KUKA KRL program: EPS_2_251825_SA27_A_20260116064105.src

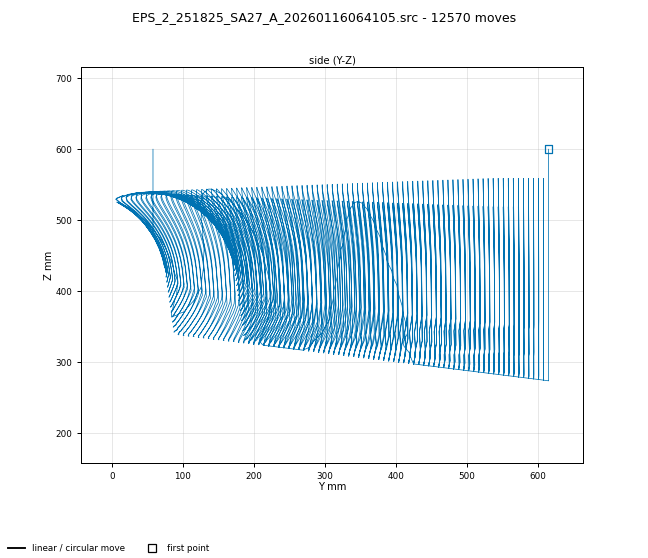
[picture p0: tool path of EPS_2_251825_SA27_A_20260116064105.src, 12570 of 12572 moves have a stored position in this frame; points joined in program order, loops and branches not executed]
&ACCESS RVP
&REL 4
&COMMENT QRS 19112012
&PARAM EDITMASK = *
DEF PART()
EXT BAS (BAS_COMMAND :IN,REAL :IN )
INT I
BAS (#INITMOV,0 )

;KUKA QRS Post kuka4.cps  Date:22-06-2017 !

File_ID=2986

QRS_PRE_INIT()

;Init var - Until changes are made in qrs_pre_init
Outlet_Square_prg=0
Inlet_1_Square_prg=0
Inlet_2_Square_prg=0
Inlet_3_Square_prg=0
Inlet_4_Square_prg=0
Inlet_5_Square_prg=0

Outlet_1={X 0.000, Y 535.490, Z 458.500, B 0.000, E1 0.000 }
Inlet_1={X 0.000, Y 538.340, Z 418.500, B 0.000, E1 212.000 }
Outlet_1_type=201
Inlet_1_type=201
;QRS#1=Sidecore dimensions
;QRS#2=200-8" PVC SDR 35
;QRS#3=200-8" PVC SDR 35
;QRS#4=
;QRS#5=
;QRS#6=
;QRS#7=
;QRS#8=
;QRS#9=12-08 PSX
;QRS#10=12-08 PSX
;QRS#11=
;QRS#12=
;QRS#13=
;QRS#14=
;QRS#15=
;QRS#16=1220x127x838 2,75'
;QRS#17=EPS Height
;QRS#18=559
;QRS#19=*
;QRS#20= UPDATED VERSION 22-06-2017
;QRS#21=*
Outlet_Square=0100
Inlet_1_Square=0100
Inlet_2_Square=0
Inlet_3_Square=0
Inlet_4_Square=0
Inlet_5_Square=0
Mill_Square=1
Outlet_Square_Prg=204
Inlet_1_Square_prg=204

QRS_INIT()

$ADVANCE=5

; T1
PTP {E1 173.63,E2 173.63}
PTP {X 0,Y 615.439,A -85,B 0,C 180,E1 173.63,E2 173.63,E3 0,E4 0,E5 0,E6 0}
QRS_SPEED_INIT()
LIN {X 0,Y 615.439,Z 600,A -85,B 0,C 180,E1 173.63,E2 173.63,E3 0,E4 0,E5 0,E6 0} C_VEL
LIN {X 0,Y 615.439,Z 283.873,A -85,B 0,C 180,E1 173.63,E2 173.63} C_VEL
LIN {X 0,Y 615.439,Z 275.692,A -85,B 0,C 180,E1 173.63,E2 173.63} C_VEL
LIN {X 0,Y 615.44,Z 273.692,A -85,B 0,C 180,E1 173.444,E2 173.444} C_VEL
LIN {X 0,Y 615.485,Z 273.687,A -85,B 0,C 180,E1 170.801,E2 170.801} C_VEL
LIN {X 0,Y 615.48,Z 273.701,A -85,B 0,C 180,E1 168.139,E2 168.139} C_VEL
LIN {X 0,Y 615.434,Z 273.695,A -85,B 0,C 180,E1 165.45,E2 165.45} C_VEL
LIN {X 0,Y 615.431,Z 273.695,A -85,B 0,C 180,E1 163.412,E2 163.412} C_VEL
LIN {X 0,Y 615.431,Z 273.695,A -85,B 0,C 180,E1 161.352,E2 161.352} C_VEL
LIN {X 0,Y 615.429,Z 273.695,A -85,B 0,C 180,E1 159.267,E2 159.267} C_VEL
LIN {X 0,Y 615.427,Z 273.695,A -85,B 0,C 180,E1 157.153,E2 157.153} C_VEL
LIN {X 0,Y 615.424,Z 273.695,A -85,B 0,C 180,E1 155.005,E2 155.005} C_VEL
LIN {X 0,Y 615.425,Z 273.695,A -85,B 0,C 180,E1 152.82,E2 152.82} C_VEL
LIN {X 0,Y 615.469,Z 273.693,A -85,B 0,C 180,E1 150.206,E2 150.206} C_VEL
LIN {X 0,Y 615.469,Z 273.699,A -85,B 0,C 180,E1 147.541,E2 147.541} C_VEL
LIN {X 0,Y 615.434,Z 273.698,A -85,B 0,C 180,E1 145.181,E2 145.181} C_VEL
LIN {X 0,Y 615.415,Z 273.698,A -85,B 0,C 180,E1 142.752,E2 142.752} C_VEL
LIN {X 0,Y 615.46,Z 273.696,A -85,B 0,C 180,E1 139.913,E2 139.913} C_VEL
LIN {X 0,Y 615.489,Z 273.697,A -85,B 0,C 180,E1 137.647,E2 137.647} C_VEL
LIN {X 0,Y 615.426,Z 273.7,A -85,B 0,C 180,E1 134.925,E2 134.925} C_VEL
LIN {X 0,Y 615.445,Z 273.7,A -85,B 0,C 180,E1 133.043,E2 133.043} C_VEL
LIN {X 0,Y 615.41,Z 273.7,A -85,B 0,C 180,E1 130.612,E2 130.612} C_VEL
LIN {X 0,Y 615.407,Z 273.7,A -85,B 0,C 180,E1 128.074,E2 128.074} C_VEL
LIN {X 0,Y 615.435,Z 273.701,A -85,B 0,C 180,E1 125.619,E2 125.619} C_VEL
LIN {X 0,Y 615.47,Z 273.704,A -85,B 0,C 180,E1 123.237,E2 123.237} C_VEL
LIN {X 0,Y 615.472,Z 273.699,A -85,B 0,C 180,E1 120.921,E2 120.921} C_VEL
LIN {X 0,Y 615.431,Z 273.697,A -85,B 0,C 180,E1 118.44,E2 118.44} C_VEL
LIN {X 0,Y 615.434,Z 273.697,A -85,B 0,C 180,E1 116.447,E2 116.447} C_VEL
LIN {X 0,Y 615.427,Z 273.697,A -85,B 0,C 180,E1 114.275,E2 114.275} C_VEL
LIN {X 0,Y 615.427,Z 273.696,A -85,B 0,C 180,E1 112.139,E2 112.139} C_VEL
LIN {X 0,Y 615.426,Z 273.695,A -85,B 0,C 180,E1 110.036,E2 110.036} C_VEL
LIN {X 0,Y 615.427,Z 273.695,A -85,B 0,C 180,E1 107.96,E2 107.96} C_VEL
LIN {X 0,Y 615.429,Z 273.695,A -85,B 0,C 180,E1 105.908,E2 105.908} C_VEL
LIN {X 0,Y 615.432,Z 273.694,A -85,B 0,C 180,E1 103.877,E2 103.877} C_VEL
LIN {X 0,Y 615.437,Z 273.693,A -85,B 0,C 180,E1 101.863,E2 101.863} C_VEL
LIN {X 0,Y 615.443,Z 273.692,A -85,B 0,C 180,E1 99.864,E2 99.864} C_VEL
LIN {X 0,Y 615.448,Z 273.692,A -85,B 0,C 180,E1 97.878,E2 97.878} C_VEL
LIN {X 0,Y 615.46,Z 273.69,A -85,B 0,C 180,E1 95.901,E2 95.901} C_VEL
LIN {X 0,Y 615.432,Z 273.694,A -85,B 0,C 180,E1 93.275,E2 93.275} C_VEL
LIN {X 0,Y 615.464,Z 273.698,A -85,B 0,C 180,E1 90.656,E2 90.656} C_VEL
LIN {X 0,Y 615.497,Z 273.69,A -85,B 0,C 180,E1 88.039,E2 88.039} C_VEL
LIN {X 0,Y 615.451,Z 273.69,A -85,B 0,C 180,E1 85.418,E2 85.418} C_VEL
LIN {X 0,Y 615.456,Z 273.689,A -85,B 0,C 180,E1 83.446,E2 83.446} C_VEL
LIN {X 0,Y 615.468,Z 273.687,A -85,B 0,C 180,E1 81.466,E2 81.466} C_VEL
LIN {X 0,Y 615.449,Z 273.689,A -85,B 0,C 180,E1 79.132,E2 79.132} C_VEL
LIN {X 0,Y 615.448,Z 273.76,A -85,B 0,C 180,E1 76.612,E2 76.612} C_VEL
LIN {X 0,Y 615.487,Z 288.561,A -85,B 0,C 180,E1 74.098,E2 74.098} C_VEL
LIN {X 0,Y 615.49,Z 304.913,A -85,B 0,C 180,E1 71.358,E2 71.358} C_VEL
LIN {X 0,Y 615.481,Z 308.156,A -85,B 0,C 180,E1 70.817,E2 70.817} C_VEL
LIN {X 0,Y 615.479,Z 414.874,A -85,B 0,C 180,E1 69.544,E2 69.544} C_VEL
LIN {X 0,Y 615.49,Z 427.341,A -85,B 0,C 180,E1 69.273,E2 69.273} C_VEL
LIN {X 0,Y 615.492,Z 439.612,A -85,B 0,C 180,E1 68.879,E2 68.879} C_VEL
LIN {X 0,Y 615.472,Z 450.84,A -85,B 0,C 180,E1 68.396,E2 68.396} C_VEL
LIN {X 0,Y 615.466,Z 462.297,A -85,B 0,C 180,E1 67.762,E2 67.762} C_VEL
LIN {X 0,Y 615.498,Z 473.358,A -85,B 0,C 180,E1 66.982,E2 66.982} C_VEL
LIN {X 0,Y 615.498,Z 482.093,A -85,B 0,C 180,E1 66.219,E2 66.219} C_VEL
LIN {X 0,Y 615.497,Z 490.274,A -85,B 0,C 180,E1 65.373,E2 65.373} C_VEL
LIN {X 0,Y 615.493,Z 497.637,A -85,B 0,C 180,E1 64.431,E2 64.431} C_VEL
LIN {X 0,Y 615.497,Z 503.202,A -85,B 0,C 180,E1 63.561,E2 63.561} C_VEL
LIN {X 0,Y 615.496,Z 508.785,A -85,B 0,C 180,E1 62.459,E2 62.459} C_VEL
LIN {X 0,Y 615.496,Z 513.017,A -85,B 0,C 180,E1 61.347,E2 61.347} C_VEL
LIN {X 0,Y 615.496,Z 516.043,A -85,B 0,C 180,E1 60.205,E2 60.205} C_VEL
LIN {X 0,Y 615.497,Z 517.96,A -85,B 0,C 180,E1 58.913,E2 58.913} C_VEL
LIN {X 0,Y 615.494,Z 518.326,A -85,B 0,C 180,E1 57.669,E2 57.669} C_VEL
LIN {X 0,Y 615.496,Z 517.367,A -85,B 0,C 180,E1 56.465,E2 56.465} C_VEL
LIN {X 0,Y 615.492,Z 514.843,A -85,B 0,C 180,E1 55.191,E2 55.191} C_VEL
LIN {X 0,Y 615.495,Z 511.661,A -85,B 0,C 180,E1 54.166,E2 54.166} C_VEL
LIN {X 0,Y 615.492,Z 506.976,A -85,B 0,C 180,E1 53.063,E2 53.063} C_VEL
LIN {X 0,Y 615.495,Z 500.7,A -85,B 0,C 180,E1 51.938,E2 51.938} C_VEL
LIN {X 0,Y 615.496,Z 493.587,A -85,B 0,C 180,E1 50.937,E2 50.937} C_VEL
LIN {X 0,Y 615.497,Z 486.114,A -85,B 0,C 180,E1 50.084,E2 50.084} C_VEL
LIN {X 0,Y 615.495,Z 476.164,A -85,B 0,C 180,E1 49.153,E2 49.153} C_VEL
LIN {X 0,Y 615.481,Z 465.87,A -85,B 0,C 180,E1 48.381,E2 48.381} C_VEL
LIN {X 0,Y 615.459,Z 454.84,A -85,B 0,C 180,E1 47.719,E2 47.719} C_VEL
LIN {X 0,Y 615.495,Z 442.203,A -85,B 0,C 180,E1 47.129,E2 47.129} C_VEL
LIN {X 0,Y 615.492,Z 430.199,A -85,B 0,C 180,E1 46.715,E2 46.715} C_VEL
LIN {X 0,Y 615.482,Z 417.178,A -85,B 0,C 180,E1 46.409,E2 46.409} C_VEL
LIN {X 0,Y 615.471,Z 395.409,A -85,B 0,C 180,E1 46.124,E2 46.124} C_VEL
LIN {X 0,Y 615.482,Z 308.164,A -85,B 0,C 180,E1 45.094,E2 45.094} C_VEL
LIN {X 0,Y 615.496,Z 291.775,A -85,B 0,C 180,E1 42.353,E2 42.353} C_VEL
LIN {X 0,Y 615.465,Z 275.402,A -85,B 0,C 180,E1 39.579,E2 39.579} C_VEL
LIN {X 0,Y 615.445,Z 273.695,A -85,B 0,C 180,E1 39.279,E2 39.279} C_VEL
LIN {X 0,Y 615.439,Z 273.692,A -85,B 0,C 180,E1 36.939,E2 36.939} C_VEL
LIN {X 0,Y 615.443,Z 273.691,A -85,B 0,C 180,E1 34.704,E2 34.704} C_VEL
LIN {X 0,Y 615.465,Z 273.69,A -85,B 0,C 180,E1 32.338,E2 32.338} C_VEL
LIN {X 0,Y 615.463,Z 273.698,A -85,B 0,C 180,E1 29.408,E2 29.408} C_VEL
LIN {X 0,Y 615.434,Z 273.697,A -85,B 0,C 180,E1 27.048,E2 27.048} C_VEL
LIN {X 0,Y 615.432,Z 273.697,A -85,B 0,C 180,E1 24.994,E2 24.994} C_VEL
LIN {X 0,Y 615.425,Z 273.697,A -85,B 0,C 180,E1 22.847,E2 22.847} C_VEL
LIN {X 0,Y 615.418,Z 273.697,A -85,B 0,C 180,E1 20.556,E2 20.556} C_VEL
LIN {X 0,Y 615.446,Z 273.696,A -85,B 0,C 180,E1 17.958,E2 17.958} C_VEL
LIN {X 0,Y 615.469,Z 273.7,A -85,B 0,C 180,E1 15.227,E2 15.227} C_VEL
LIN {X 0,Y 615.409,Z 273.699,A -85,B 0,C 180,E1 12.532,E2 12.532} C_VEL
LIN {X 0,Y 615.408,Z 273.7,A -85,B 0,C 180,E1 10.528,E2 10.528} C_VEL
LIN {X 0,Y 615.41,Z 273.7,A -85,B 0,C 180,E1 8.538,E2 8.538} C_VEL
LIN {X 0,Y 615.416,Z 273.699,A -85,B 0,C 180,E1 6.557,E2 6.557} C_VEL
LIN {X 0,Y 615.423,Z 273.699,A -85,B 0,C 180,E1 4.585,E2 4.585} C_VEL
LIN {X 0,Y 615.434,Z 273.697,A -85,B 0,C 180,E1 2.618,E2 2.618} C_VEL
LIN {X 0,Y 615.442,Z 273.697,A -85,B 0,C 180,E1 0.654,E2 0.654} C_VEL
LIN {X 0,Y 615.417,Z 273.697,A -85,B 0,C 180,E1 -1.963,E2 -1.963} C_VEL
LIN {X 0,Y 615.419,Z 273.697,A -85,B 0,C 180,E1 -3.929,E2 -3.929} C_VEL
LIN {X 0,Y 615.426,Z 273.695,A -85,B 0,C 180,E1 -5.899,E2 -5.899} C_VEL
LIN {X 0,Y 615.432,Z 273.694,A -85,B 0,C 180,E1 -7.876,E2 -7.876} C_VEL
LIN {X 0,Y 615.438,Z 273.693,A -85,B 0,C 180,E1 -9.863,E2 -9.863} C_VEL
LIN {X 0,Y 615.443,Z 273.692,A -85,B 0,C 180,E1 -11.862,E2 -11.862} C_VEL
LIN {X 0,Y 615.444,Z 273.692,A -85,B 0,C 180,E1 -13.941,E2 -13.941} C_VEL
LIN {X 0,Y 615.454,Z 273.69,A -85,B 0,C 180,E1 -15.906,E2 -15.906} C_VEL
LIN {X 0,Y 615.456,Z 273.689,A -85,B 0,C 180,E1 -17.958,E2 -17.958} C_VEL
LIN {X 0,Y 615.457,Z 273.689,A -85,B 0,C 180,E1 -20.034,E2 -20.034} C_VEL
LIN {X 0,Y 615.445,Z 273.691,A -85,B 0,C 180,E1 -22.351,E2 -22.351} C_VEL
LIN {X 0,Y 615.452,Z 273.689,A -85,B 0,C 180,E1 -24.274,E2 -24.274} C_VEL
LIN {X 0,Y 615.448,Z 273.69,A -85,B 0,C 180,E1 -26.446,E2 -26.446} C_VEL
LIN {X 0,Y 615.449,Z 273.691,A -85,B 0,C 180,E1 -28.66,E2 -28.66} C_VEL
LIN {X 0,Y 615.464,Z 273.696,A -85,B 0,C 180,E1 -31.093,E2 -31.093} C_VEL
LIN {X 0,Y 615.494,Z 273.684,A -85,B 0,C 180,E1 -34.022,E2 -34.022} C_VEL
LIN {X 0,Y 615.477,Z 273.684,A -85,B 0,C 180,E1 -36.426,E2 -36.426} C_VEL
LIN {X 0,Y 615.461,Z 273.692,A -85,B 0,C 180,E1 -39.067,E2 -39.067} C_VEL
LIN {X 0,Y 615.477,Z 273.699,A -85,B 0,C 180,E1 -41.475,E2 -41.475} C_VEL
LIN {X 0,Y 615.484,Z 273.688,A -85,B 0,C 180,E1 -44.15,E2 -44.15} C_VEL
LIN {X 0,Y 615.47,Z 273.686,A -85,B 0,C 180,E1 -46.955,E2 -46.955} C_VEL
LIN {X 0,Y 615.471,Z 273.693,A -85,B 0,C 180,E1 -49.399,E2 -49.399} C_VEL
LIN {X 0,Y 615.489,Z 273.697,A -85,B 0,C 180,E1 -51.988,E2 -51.988} C_VEL
LIN {X 0,Y 615.476,Z 273.689,A -85,B 0,C 180,E1 -54.389,E2 -54.389} C_VEL
LIN {X 0,Y 615.483,Z 273.683,A -85,B 0,C 180,E1 -56.769,E2 -56.769} C_VEL
LIN {X 0,Y 615.483,Z 273.682,A -85,B 0,C 180,E1 -59.085,E2 -59.085} C_VEL
LIN {X 0,Y 615.477,Z 273.69,A -85,B 0,C 180,E1 -61.552,E2 -61.552} C_VEL
LIN {X 0,Y 615.481,Z 273.696,A -85,B 0,C 180,E1 -64.288,E2 -64.288} C_VEL
LIN {X 0,Y 615.489,Z 273.681,A -85,B 0,C 180,E1 -67.16,E2 -67.16} C_VEL
LIN {X 0,Y 615.487,Z 273.766,A -85,B 0,C 180,E1 -67.439,E2 -67.439} C_VEL
LIN {X 0,Y 615.456,Z 293.719,A -85,B 0,C 180,E1 -70.144,E2 -70.144} C_VEL
LIN {X 0,Y 615.472,Z 313.103,A -85,B 0,C 180,E1 -72.733,E2 -72.733} C_VEL
LIN {X 0,Y 615.493,Z 334.935,A -85,B 0,C 180,E1 -75.609,E2 -75.609} C_VEL
LIN {X 0,Y 615.471,Z 346.492,A -85,B 0,C 180,E1 -77.116,E2 -77.116} C_VEL
LIN {X 0,Y 615.457,Z 455.001,A -85,B 0,C 180,E1 -78.413,E2 -78.413} C_VEL
LIN {X 0,Y 615.456,Z 467.457,A -85,B 0,C 180,E1 -78.684,E2 -78.684} C_VEL
LIN {X 0,Y 615.483,Z 480.688,A -85,B 0,C 180,E1 -79.116,E2 -79.116} C_VEL
LIN {X 0,Y 615.492,Z 492.532,A -85,B 0,C 180,E1 -79.642,E2 -79.642} C_VEL
LIN {X 0,Y 615.483,Z 504.039,A -85,B 0,C 180,E1 -80.307,E2 -80.307} C_VEL
LIN {X 0,Y 615.499,Z 514.376,A -85,B 0,C 180,E1 -81.053,E2 -81.053} C_VEL
LIN {X 0,Y 615.497,Z 522.719,A -85,B 0,C 180,E1 -81.797,E2 -81.797} C_VEL
LIN {X 0,Y 615.498,Z 530.629,A -85,B 0,C 180,E1 -82.622,E2 -82.622} C_VEL
LIN {X 0,Y 615.491,Z 538.221,A -85,B 0,C 180,E1 -83.611,E2 -83.611} C_VEL
LIN {X 0,Y 615.498,Z 545.218,A -85,B 0,C 180,E1 -84.761,E2 -84.761} C_VEL
LIN {X 0,Y 615.493,Z 549.862,A -85,B 0,C 180,E1 -85.746,E2 -85.746} C_VEL
LIN {X 0,Y 615.494,Z 553.406,A -85,B 0,C 180,E1 -86.729,E2 -86.729} C_VEL
LIN {X 0,Y 615.497,Z 555.239,A -85,B 0,C 180,E1 -87.384,E2 -87.384} C_VEL
LIN {X 0,Y 615.497,Z 556.612,A -85,B 0,C 180,E1 -88.039,E2 -88.039} C_VEL
LIN {X 0,Y 615.496,Z 558.175,A -85,B 0,C 180,E1 -89.348,E2 -89.348} C_VEL
LIN {X 0,Y 615.494,Z 558.389,A -85,B 0,C 180,E1 -90.002,E2 -90.002} C_VEL
LIN {X 0,Y 615.495,Z 557.578,A -85,B 0,C 180,E1 -91.311,E2 -91.311} C_VEL
LIN {X 0,Y 615.497,Z 556.605,A -85,B 0,C 180,E1 -91.965,E2 -91.965} C_VEL
LIN {X 0,Y 615.497,Z 555.228,A -85,B 0,C 180,E1 -92.62,E2 -92.62} C_VEL
LIN {X 0,Y 615.496,Z 552.343,A -85,B 0,C 180,E1 -93.603,E2 -93.603} C_VEL
LIN {X 0,Y 615.498,Z 548.434,A -85,B 0,C 180,E1 -94.586,E2 -94.586} C_VEL
LIN {X 0,Y 615.499,Z 543.395,A -85,B 0,C 180,E1 -95.571,E2 -95.571} C_VEL
LIN {X 0,Y 615.49,Z 536.913,A -85,B 0,C 180,E1 -96.578,E2 -96.578} C_VEL
LIN {X 0,Y 615.497,Z 529.118,A -85,B 0,C 180,E1 -97.547,E2 -97.547} C_VEL
LIN {X 0,Y 615.498,Z 519.239,A -85,B 0,C 180,E1 -98.538,E2 -98.538} C_VEL
LIN {X 0,Y 615.495,Z 508.845,A -85,B 0,C 180,E1 -99.366,E2 -99.366} C_VEL
LIN {X 0,Y 615.482,Z 498.551,A -85,B 0,C 180,E1 -100.03,E2 -100.03} C_VEL
LIN {X 0,Y 615.495,Z 487.113,A -85,B 0,C 180,E1 -100.617,E2 -100.617} C_VEL
LIN {X 0,Y 615.466,Z 475.331,A -85,B 0,C 180,E1 -101.079,E2 -101.079} C_VEL
LIN {X 0,Y 615.455,Z 462.187,A -85,B 0,C 180,E1 -101.445,E2 -101.445} C_VEL
LIN {X 0,Y 615.461,Z 448.837,A -85,B 0,C 180,E1 -101.675,E2 -101.675} C_VEL
LIN {X 0,Y 615.471,Z 346.459,A -85,B 0,C 180,E1 -102.888,E2 -102.888} C_VEL
LIN {X 0,Y 615.455,Z 325.982,A -85,B 0,C 180,E1 -105.567,E2 -105.567} C_VEL
LIN {X 0,Y 615.481,Z 305.471,A -85,B 0,C 180,E1 -108.282,E2 -108.282} C_VEL
LIN {X 0,Y 615.468,Z 283.338,A -85,B 0,C 180,E1 -111.258,E2 -111.258} C_VEL
LIN {X 0,Y 615.489,Z 273.682,A -85,B 0,C 180,E1 -112.594,E2 -112.594} C_VEL
LIN {X 0,Y 615.485,Z 273.681,A -85,B 0,C 180,E1 -114.992,E2 -114.992} C_VEL
LIN {X 0,Y 615.481,Z 273.7,A -85,B 0,C 180,E1 -117.916,E2 -117.916} C_VEL
LIN {X 0,Y 615.492,Z 273.698,A -85,B 0,C 180,E1 -120.16,E2 -120.16} C_VEL
LIN {X 0,Y 615.479,Z 273.692,A -85,B 0,C 180,E1 -122.458,E2 -122.458} C_VEL
LIN {X 0,Y 615.478,Z 273.686,A -85,B 0,C 180,E1 -124.815,E2 -124.815} C_VEL
LIN {X 0,Y 615.49,Z 273.68,A -85,B 0,C 180,E1 -127.242,E2 -127.242} C_VEL
LIN {X 0,Y 615.484,Z 273.695,A -85,B 0,C 180,E1 -130.088,E2 -130.088} C_VEL
LIN {X 0,Y 615.499,Z 273.7,A -85,B 0,C 180,E1 -132.351,E2 -132.351} C_VEL
LIN {X 0,Y 615.472,Z 273.687,A -85,B 0,C 180,E1 -135.069,E2 -135.069} C_VEL
LIN {X 0,Y 615.482,Z 273.686,A -85,B 0,C 180,E1 -137.919,E2 -137.919} C_VEL
LIN {X 0,Y 615.483,Z 273.693,A -85,B 0,C 180,E1 -140.249,E2 -140.249} C_VEL
LIN {X 0,Y 615.467,Z 273.692,A -85,B 0,C 180,E1 -143.064,E2 -143.064} C_VEL
LIN {X 0,Y 615.466,Z 273.689,A -85,B 0,C 180,E1 -145.3,E2 -145.3} C_VEL
LIN {X 0,Y 615.476,Z 273.683,A -85,B 0,C 180,E1 -147.669,E2 -147.669} C_VEL
LIN {X 0,Y 615.486,Z 273.696,A -85,B 0,C 180,E1 -150.594,E2 -150.594} C_VEL
LIN {X 0,Y 615.488,Z 273.698,A -85,B 0,C 180,E1 -152.952,E2 -152.952} C_VEL
LIN {X 0,Y 615.463,Z 273.687,A -85,B 0,C 180,E1 -155.727,E2 -155.727} C_VEL
LIN {X 0,Y 615.488,Z 273.688,A -85,B 0,C 180,E1 -158.568,E2 -158.568} C_VEL
LIN {X 0,Y 615.466,Z 273.695,A -85,B 0,C 180,E1 -161.396,E2 -161.396} C_VEL
LIN {X 0,Y 615.464,Z 273.686,A -85,B 0,C 180,E1 -164.094,E2 -164.094} C_VEL
LIN {X 0,Y 615.491,Z 273.689,A -85,B 0,C 180,E1 -166.799,E2 -166.799} C_VEL
LIN {X 0,Y 615.473,Z 273.697,A -85,B 0,C 180,E1 -169.473,E2 -169.473} C_VEL
LIN {X 0,Y 615.45,Z 273.69,A -85,B 0,C 180,E1 -172.124,E2 -172.124} C_VEL
LIN {X 0,Y 615.486,Z 273.685,A -85,B 0,C 180,E1 -174.759,E2 -174.759} C_VEL
LIN {X 0,Y 615.497,Z 273.699,A -85,B 0,C 180,E1 -177.382,E2 -177.382} C_VEL
LIN {X 0,Y 615.448,Z 273.695,A -85,B 0,C 180,E1 -180,E2 -180} C_VEL
LIN {X 0,Y 615.454,Z 273.696,A -85,B 0,C 180,E1 -181.963,E2 -181.963} C_VEL
LIN {X 0,Y 615.459,Z 273.697,A -85,B 0,C 180,E1 -183.929,E2 -183.929} C_VEL
LIN {X 0,Y 615.466,Z 273.698,A -85,B 0,C 180,E1 -185.899,E2 -185.899} C_VEL
LIN {X 0,Y 615.44,Z 273.692,A -85,B 0,C 180,E1 -186.556,E2 -186.556} C_VEL
LIN {X 0,Y 614.8,Z 273.837,A -85,B 0,C 180,E1 -187.102,E2 -187.102} C_VEL
LIN {X 0,Y 611.989,Z 274.252,A -85,B 0,C 180,E1 -187.988,E2 -187.988} C_VEL
LIN {X 0,Y 609.593,Z 274.561,A -85,B 0,C 180,E1 -188.701,E2 -188.701} C_VEL
LIN {X 0,Y 608.548,Z 274.68,A -85,B 0,C 180,E1 -189.25,E2 -189.25} C_VEL
LIN {X 0,Y 608.455,Z 274.69,A -85,B 0,C 180,E1 -189.437,E2 -189.437} C_VEL
LIN {X 0,Y 608.445,Z 274.695,A -85,B 0,C 180,E1 -192,E2 -192} C_VEL
LIN {X 0,Y 608.405,Z 274.693,A -85,B 0,C 180,E1 -194.722,E2 -194.722} C_VEL
LIN {X 0,Y 608.435,Z 274.693,A -85,B 0,C 180,E1 -197.477,E2 -197.477} C_VEL
LIN {X 0,Y 608.437,Z 274.694,A -85,B 0,C 180,E1 -200.275,E2 -200.275} C_VEL
LIN {X 0,Y 608.415,Z 274.695,A -85,B 0,C 180,E1 -202.47,E2 -202.47} C_VEL
LIN {X 0,Y 608.42,Z 274.693,A -85,B 0,C 180,E1 -204.573,E2 -204.573} C_VEL
LIN {X 0,Y 608.406,Z 274.692,A -85,B 0,C 180,E1 -207.197,E2 -207.197} C_VEL
LIN {X 0,Y 608.46,Z 274.693,A -85,B 0,C 180,E1 -209.973,E2 -209.973} C_VEL
LIN {X 0,Y 608.417,Z 274.693,A -85,B 0,C 180,E1 -212.882,E2 -212.882} C_VEL
LIN {X 0,Y 608.394,Z 274.694,A -85,B 0,C 180,E1 -215.281,E2 -215.281} C_VEL
LIN {X 0,Y 608.446,Z 274.696,A -85,B 0,C 180,E1 -218.239,E2 -218.239} C_VEL
LIN {X 0,Y 608.432,Z 274.698,A -85,B 0,C 180,E1 -220.328,E2 -220.328} C_VEL
LIN {X 0,Y 608.401,Z 274.696,A -85,B 0,C 180,E1 -222.965,E2 -222.965} C_VEL
LIN {X 0,Y 608.399,Z 274.695,A -85,B 0,C 180,E1 -225.2,E2 -225.2} C_VEL
LIN {X 0,Y 608.408,Z 274.696,A -85,B 0,C 180,E1 -227.037,E2 -227.037} C_VEL
LIN {X 0,Y 608.432,Z 274.697,A -85,B 0,C 180,E1 -228.822,E2 -228.822} C_VEL
LIN {X 0,Y 608.387,Z 274.696,A -85,B 0,C 180,E1 -231.406,E2 -231.406} C_VEL
LIN {X 0,Y 608.42,Z 274.696,A -85,B 0,C 180,E1 -233.083,E2 -233.083} C_VEL
LIN {X 0,Y 608.389,Z 274.695,A -85,B 0,C 180,E1 -235.526,E2 -235.526} C_VEL
LIN {X 0,Y 608.403,Z 274.693,A -85,B 0,C 180,E1 -237.902,E2 -237.902} C_VEL
LIN {X 0,Y 608.404,Z 274.693,A -85,B 0,C 180,E1 -240.217,E2 -240.217} C_VEL
LIN {X 0,Y 608.452,Z 274.694,A -85,B 0,C 180,E1 -242.798,E2 -242.798} C_VEL
LIN {X 0,Y 608.427,Z 274.694,A -85,B 0,C 180,E1 -245.427,E2 -245.427} C_VEL
LIN {X 0,Y 608.417,Z 274.691,A -85,B 0,C 180,E1 -248.306,E2 -248.306} C_VEL
LIN {X 0,Y 608.404,Z 274.693,A -85,B 0,C 180,E1 -250.427,E2 -250.427} C_VEL
LIN {X 0,Y 608.406,Z 274.693,A -85,B 0,C 180,E1 -252.521,E2 -252.521} C_VEL
LIN {X 0,Y 608.47,Z 274.696,A -85,B 0,C 180,E1 -255.278,E2 -255.278} C_VEL
LIN {X 0,Y 608.43,Z 274.691,A -85,B 0,C 180,E1 -257.998,E2 -257.998} C_VEL
LIN {X 0,Y 608.424,Z 274.692,A -85,B 0,C 180,E1 -260.021,E2 -260.021} C_VEL
LIN {X 0,Y 608.421,Z 274.692,A -85,B 0,C 180,E1 -262.031,E2 -262.031} C_VEL
LIN {X 0,Y 608.438,Z 274.691,A -85,B 0,C 180,E1 -264.031,E2 -264.031} C_VEL
LIN {X 0,Y 608.404,Z 274.693,A -85,B 0,C 180,E1 -266.687,E2 -266.687} C_VEL
LIN {X 0,Y 608.46,Z 274.692,A -85,B 0,C 180,E1 -269.336,E2 -269.336} C_VEL
LIN {X 0,Y 608.465,Z 274.691,A -85,B 0,C 180,E1 -271.983,E2 -271.983} C_VEL
LIN {X 0,Y 608.419,Z 274.691,A -85,B 0,C 180,E1 -274.635,E2 -274.635} C_VEL
LIN {X 0,Y 608.435,Z 274.689,A -85,B 0,C 180,E1 -276.63,E2 -276.63} C_VEL
LIN {X 0,Y 608.437,Z 274.689,A -85,B 0,C 180,E1 -278.634,E2 -278.634} C_VEL
LIN {X 0,Y 608.421,Z 274.691,A -85,B 0,C 180,E1 -280.931,E2 -280.931} C_VEL
LIN {X 0,Y 608.455,Z 274.79,A -85,B 0,C 180,E1 -283.332,E2 -283.332} C_VEL
LIN {X 0,Y 608.493,Z 289.89,A -85,B 0,C 180,E1 -285.917,E2 -285.917} C_VEL
LIN {X 0,Y 608.471,Z 306.465,A -85,B 0,C 180,E1 -288.715,E2 -288.715} C_VEL
LIN {X 0,Y 608.448,Z 308.354,A -85,B 0,C 180,E1 -289.031,E2 -289.031} C_VEL
LIN {X 0,Y 608.531,Z 415.658,A -85,B 0,C 180,E1 -290.334,E2 -290.334} C_VEL
LIN {X 0,Y 608.552,Z 429.268,A -85,B 0,C 180,E1 -290.646,E2 -290.646} C_VEL
LIN {X 0,Y 608.526,Z 441.594,A -85,B 0,C 180,E1 -291.064,E2 -291.064} C_VEL
LIN {X 0,Y 608.472,Z 453.291,A -85,B 0,C 180,E1 -291.599,E2 -291.599} C_VEL
LIN {X 0,Y 608.462,Z 464.004,A -85,B 0,C 180,E1 -292.223,E2 -292.223} C_VEL
LIN {X 0,Y 608.499,Z 474.949,A -85,B 0,C 180,E1 -293.019,E2 -293.019} C_VEL
LIN {X 0,Y 608.471,Z 482.15,A -85,B 0,C 180,E1 -293.66,E2 -293.66} C_VEL
LIN {X 0,Y 608.471,Z 490.85,A -85,B 0,C 180,E1 -294.566,E2 -294.566} C_VEL
LIN {X 0,Y 608.445,Z 498.138,A -85,B 0,C 180,E1 -295.507,E2 -295.507} C_VEL
LIN {X 0,Y 608.439,Z 504.819,A -85,B 0,C 180,E1 -296.585,E2 -296.585} C_VEL
LIN {X 0,Y 608.435,Z 509.408,A -85,B 0,C 180,E1 -297.514,E2 -297.514} C_VEL
LIN {X 0,Y 608.426,Z 513.564,A -85,B 0,C 180,E1 -298.611,E2 -298.611} C_VEL
LIN {X 0,Y 608.437,Z 517.043,A -85,B 0,C 180,E1 -299.966,E2 -299.966} C_VEL
LIN {X 0,Y 608.441,Z 518.701,A -85,B 0,C 180,E1 -301.266,E2 -301.266} C_VEL
LIN {X 0,Y 608.421,Z 518.896,A -85,B 0,C 180,E1 -302.516,E2 -302.516} C_VEL
LIN {X 0,Y 608.421,Z 517.706,A -85,B 0,C 180,E1 -303.727,E2 -303.727} C_VEL
LIN {X 0,Y 608.421,Z 515.255,A -85,B 0,C 180,E1 -304.901,E2 -304.901} C_VEL
LIN {X 0,Y 608.442,Z 511.423,A -85,B 0,C 180,E1 -306.087,E2 -306.087} C_VEL
LIN {X 0,Y 608.432,Z 506.693,A -85,B 0,C 180,E1 -307.153,E2 -307.153} C_VEL
LIN {X 0,Y 608.451,Z 500.457,A -85,B 0,C 180,E1 -308.238,E2 -308.238} C_VEL
LIN {X 0,Y 608.447,Z 492.74,A -85,B 0,C 180,E1 -309.294,E2 -309.294} C_VEL
LIN {X 0,Y 608.476,Z 484.621,A -85,B 0,C 180,E1 -310.187,E2 -310.187} C_VEL
LIN {X 0,Y 608.493,Z 476.444,A -85,B 0,C 180,E1 -310.948,E2 -310.948} C_VEL
LIN {X 0,Y 608.469,Z 467.005,A -85,B 0,C 180,E1 -311.669,E2 -311.669} C_VEL
LIN {X 0,Y 608.458,Z 456.235,A -85,B 0,C 180,E1 -312.334,E2 -312.334} C_VEL
LIN {X 0,Y 608.52,Z 443.489,A -85,B 0,C 180,E1 -312.947,E2 -312.947} C_VEL
LIN {X 0,Y 608.528,Z 431.407,A -85,B 0,C 180,E1 -313.383,E2 -313.383} C_VEL
LIN {X 0,Y 608.532,Z 418.152,A -85,B 0,C 180,E1 -313.709,E2 -313.709} C_VEL
LIN {X 0,Y 608.53,Z 400.638,A -85,B 0,C 180,E1 -313.953,E2 -313.953} C_VEL
LIN {X 0,Y 608.454,Z 308.38,A -85,B 0,C 180,E1 -315.054,E2 -315.054} C_VEL
LIN {X 0,Y 608.49,Z 291.255,A -85,B 0,C 180,E1 -317.941,E2 -317.941} C_VEL
LIN {X 0,Y 608.467,Z 275.154,A -85,B 0,C 180,E1 -320.695,E2 -320.695} C_VEL
LIN {X 0,Y 608.438,Z 274.691,A -85,B 0,C 180,E1 -320.816,E2 -320.816} C_VEL
LIN {X 0,Y 608.411,Z 274.692,A -85,B 0,C 180,E1 -323.082,E2 -323.082} C_VEL
LIN {X 0,Y 608.442,Z 274.689,A -85,B 0,C 180,E1 -325.529,E2 -325.529} C_VEL
LIN {X 0,Y 608.45,Z 274.692,A -85,B 0,C 180,E1 -327.904,E2 -327.904} C_VEL
LIN {X 0,Y 608.477,Z 274.693,A -85,B 0,C 180,E1 -330.221,E2 -330.221} C_VEL
LIN {X 0,Y 608.398,Z 274.694,A -85,B 0,C 180,E1 -333.223,E2 -333.223} C_VEL
LIN {X 0,Y 608.403,Z 274.693,A -85,B 0,C 180,E1 -335.427,E2 -335.427} C_VEL
LIN {X 0,Y 608.448,Z 274.696,A -85,B 0,C 180,E1 -338.308,E2 -338.308} C_VEL
LIN {X 0,Y 608.405,Z 274.693,A -85,B 0,C 180,E1 -341.284,E2 -341.284} C_VEL
LIN {X 0,Y 608.407,Z 274.694,A -85,B 0,C 180,E1 -343.905,E2 -343.905} C_VEL
LIN {X 0,Y 608.438,Z 274.7,A -85,B 0,C 180,E1 -346.643,E2 -346.643} C_VEL
LIN {X 0,Y 608.396,Z 274.695,A -85,B 0,C 180,E1 -349.349,E2 -349.349} C_VEL
LIN {X 0,Y 608.391,Z 274.696,A -85,B 0,C 180,E1 -351.363,E2 -351.363} C_VEL
LIN {X 0,Y 608.416,Z 274.693,A -85,B 0,C 180,E1 -353.367,E2 -353.367} C_VEL
LIN {X 0,Y 608.396,Z 274.696,A -85,B 0,C 180,E1 -355.362,E2 -355.362} C_VEL
LIN {X 0,Y 608.426,Z 274.692,A -85,B 0,C 180,E1 -357.352,E2 -357.352} C_VEL
LIN {X 0,Y 608.405,Z 274.693,A -85,B 0,C 180,E1 -360,E2 -360} C_VEL
LIN {X 0,Y 608.445,Z 274.694,A -85,B 0,C 180,E1 -362.648,E2 -362.648} C_VEL
LIN {X 0,Y 608.455,Z 274.692,A -85,B 0,C 180,E1 -365.302,E2 -365.302} C_VEL
LIN {X 0,Y 608.423,Z 274.69,A -85,B 0,C 180,E1 -367.968,E2 -367.968} C_VEL
LIN {X 0,Y 608.407,Z 274.692,A -85,B 0,C 180,E1 -369.978,E2 -369.978} C_VEL
LIN {X 0,Y 608.416,Z 274.691,A -85,B 0,C 180,E1 -372.001,E2 -372.001} C_VEL
LIN {X 0,Y 608.411,Z 274.692,A -85,B 0,C 180,E1 -374.039,E2 -374.039} C_VEL
LIN {X 0,Y 608.42,Z 274.692,A -85,B 0,C 180,E1 -376.535,E2 -376.535} C_VEL
LIN {X 0,Y 608.44,Z 274.693,A -85,B 0,C 180,E1 -378.87,E2 -378.87} C_VEL
LIN {X 0,Y 608.458,Z 274.69,A -85,B 0,C 180,E1 -381.692,E2 -381.692} C_VEL
LIN {X 0,Y 608.419,Z 274.691,A -85,B 0,C 180,E1 -384.573,E2 -384.573} C_VEL
LIN {X 0,Y 608.456,Z 274.695,A -85,B 0,C 180,E1 -387.215,E2 -387.215} C_VEL
LIN {X 0,Y 608.465,Z 274.687,A -85,B 0,C 180,E1 -389.982,E2 -389.982} C_VEL
LIN {X 0,Y 608.434,Z 274.691,A -85,B 0,C 180,E1 -392.881,E2 -392.881} C_VEL
LIN {X 0,Y 608.435,Z 274.696,A -85,B 0,C 180,E1 -395.278,E2 -395.278} C_VEL
LIN {X 0,Y 608.46,Z 274.687,A -85,B 0,C 180,E1 -398.248,E2 -398.248} C_VEL
LIN {X 0,Y 608.434,Z 274.692,A -85,B 0,C 180,E1 -401.178,E2 -401.178} C_VEL
LIN {X 0,Y 608.453,Z 274.691,A -85,B 0,C 180,E1 -403.314,E2 -403.314} C_VEL
LIN {X 0,Y 608.466,Z 274.689,A -85,B 0,C 180,E1 -406.137,E2 -406.137} C_VEL
LIN {X 0,Y 608.45,Z 274.687,A -85,B 0,C 180,E1 -408.829,E2 -408.829} C_VEL
LIN {X 0,Y 608.465,Z 274.695,A -85,B 0,C 180,E1 -411.76,E2 -411.76} C_VEL
LIN {X 0,Y 608.459,Z 274.696,A -85,B 0,C 180,E1 -413.953,E2 -413.953} C_VEL
LIN {X 0,Y 608.459,Z 274.69,A -85,B 0,C 180,E1 -416.334,E2 -416.334} C_VEL
LIN {X 0,Y 608.463,Z 274.686,A -85,B 0,C 180,E1 -418.73,E2 -418.73} C_VEL
LIN {X 0,Y 608.465,Z 274.687,A -85,B 0,C 180,E1 -421.382,E2 -421.382} C_VEL
LIN {X 0,Y 608.439,Z 274.698,A -85,B 0,C 180,E1 -423.969,E2 -423.969} C_VEL
LIN {X 0,Y 608.463,Z 274.696,A -85,B 0,C 180,E1 -426.159,E2 -426.159} C_VEL
LIN {X 0,Y 608.502,Z 274.849,A -85,B 0,C 180,E1 -427.316,E2 -427.316} C_VEL
LIN {X 0,Y 608.524,Z 292.435,A -85,B 0,C 180,E1 -429.732,E2 -429.732} C_VEL
LIN {X 0,Y 608.51,Z 311.85,A -85,B 0,C 180,E1 -432.355,E2 -432.355} C_VEL
LIN {X 0,Y 608.495,Z 332.56,A -85,B 0,C 180,E1 -435.112,E2 -435.112} C_VEL
LIN {X 0,Y 608.465,Z 346.718,A -85,B 0,C 180,E1 -436.976,E2 -436.976} C_VEL
LIN {X 0,Y 608.521,Z 455.11,A -85,B 0,C 180,E1 -438.279,E2 -438.279} C_VEL
LIN {X 0,Y 608.491,Z 468.324,A -85,B 0,C 180,E1 -438.574,E2 -438.574} C_VEL
LIN {X 0,Y 608.509,Z 480.687,A -85,B 0,C 180,E1 -438.984,E2 -438.984} C_VEL
LIN {X 0,Y 608.514,Z 492.69,A -85,B 0,C 180,E1 -439.522,E2 -439.522} C_VEL
LIN {X 0,Y 608.471,Z 504.241,A -85,B 0,C 180,E1 -440.194,E2 -440.194} C_VEL
LIN {X 0,Y 608.484,Z 514.629,A -85,B 0,C 180,E1 -440.949,E2 -440.949} C_VEL
LIN {X 0,Y 608.475,Z 523.03,A -85,B 0,C 180,E1 -441.702,E2 -441.702} C_VEL
LIN {X 0,Y 608.47,Z 530.983,A -85,B 0,C 180,E1 -442.537,E2 -442.537} C_VEL
LIN {X 0,Y 608.435,Z 538.309,A -85,B 0,C 180,E1 -443.488,E2 -443.488} C_VEL
LIN {X 0,Y 608.45,Z 543.88,A -85,B 0,C 180,E1 -444.368,E2 -444.368} C_VEL
LIN {X 0,Y 608.432,Z 548.961,A -85,B 0,C 180,E1 -445.365,E2 -445.365} C_VEL
LIN {X 0,Y 608.449,Z 552.904,A -85,B 0,C 180,E1 -446.36,E2 -446.36} C_VEL
LIN {X 0,Y 608.425,Z 555.815,A -85,B 0,C 180,E1 -447.354,E2 -447.354} C_VEL
LIN {X 0,Y 608.442,Z 557.205,A -85,B 0,C 180,E1 -448.016,E2 -448.016} C_VEL
LIN {X 0,Y 608.438,Z 558.785,A -85,B 0,C 180,E1 -449.34,E2 -449.34} C_VEL
LIN {X 0,Y 608.434,Z 559,A -85,B 0,C 180,E1 -450.002,E2 -450.002} C_VEL
LIN {X 0,Y 608.448,Z 558.181,A -85,B 0,C 180,E1 -451.326,E2 -451.326} C_VEL
LIN {X 0,Y 608.442,Z 557.198,A -85,B 0,C 180,E1 -451.988,E2 -451.988} C_VEL
LIN {X 0,Y 608.425,Z 555.804,A -85,B 0,C 180,E1 -452.65,E2 -452.65} C_VEL
LIN {X 0,Y 608.449,Z 552.89,A -85,B 0,C 180,E1 -453.644,E2 -453.644} C_VEL
LIN {X 0,Y 608.432,Z 548.942,A -85,B 0,C 180,E1 -454.64,E2 -454.64} C_VEL
LIN {X 0,Y 608.437,Z 542.866,A -85,B 0,C 180,E1 -455.803,E2 -455.803} C_VEL
LIN {X 0,Y 608.462,Z 536.222,A -85,B 0,C 180,E1 -456.801,E2 -456.801} C_VEL
LIN {X 0,Y 608.456,Z 527.975,A -85,B 0,C 180,E1 -457.802,E2 -457.802} C_VEL
LIN {X 0,Y 608.477,Z 517.58,A -85,B 0,C 180,E1 -458.805,E2 -458.805} C_VEL
LIN {X 0,Y 608.488,Z 506.725,A -85,B 0,C 180,E1 -459.642,E2 -459.642} C_VEL
LIN {X 0,Y 608.492,Z 495.746,A -85,B 0,C 180,E1 -460.314,E2 -460.314} C_VEL
LIN {X 0,Y 608.534,Z 483.807,A -85,B 0,C 180,E1 -460.888,E2 -460.888} C_VEL
LIN {X 0,Y 608.507,Z 471.836,A -85,B 0,C 180,E1 -461.325,E2 -461.325} C_VEL
LIN {X 0,Y 608.508,Z 459.438,A -85,B 0,C 180,E1 -461.641,E2 -461.641} C_VEL
LIN {X 0,Y 608.532,Z 443.616,A -85,B 0,C 180,E1 -461.873,E2 -461.873} C_VEL
LIN {X 0,Y 608.508,Z 347.033,A -85,B 0,C 180,E1 -463.017,E2 -463.017} C_VEL
LIN {X 0,Y 608.468,Z 344.176,A -85,B 0,C 180,E1 -463.358,E2 -463.358} C_VEL
LIN {X 0,Y 608.473,Z 324.76,A -85,B 0,C 180,E1 -465.922,E2 -465.922} C_VEL
LIN {X 0,Y 608.527,Z 303.774,A -85,B 0,C 180,E1 -468.731,E2 -468.731} C_VEL
LIN {X 0,Y 608.559,Z 283.34,A -85,B 0,C 180,E1 -471.511,E2 -471.511} C_VEL
LIN {X 0,Y 608.462,Z 274.687,A -85,B 0,C 180,E1 -472.715,E2 -472.715} C_VEL
LIN {X 0,Y 608.443,Z 274.689,A -85,B 0,C 180,E1 -475.302,E2 -475.302} C_VEL
LIN {X 0,Y 608.446,Z 274.691,A -85,B 0,C 180,E1 -477.518,E2 -477.518} C_VEL
LIN {X 0,Y 608.464,Z 274.695,A -85,B 0,C 180,E1 -479.971,E2 -479.971} C_VEL
LIN {X 0,Y 608.453,Z 274.687,A -85,B 0,C 180,E1 -482.88,E2 -482.88} C_VEL
LIN {X 0,Y 608.435,Z 274.689,A -85,B 0,C 180,E1 -485.278,E2 -485.278} C_VEL
LIN {X 0,Y 608.469,Z 274.687,A -85,B 0,C 180,E1 -487.746,E2 -487.746} C_VEL
LIN {X 0,Y 608.448,Z 274.699,A -85,B 0,C 180,E1 -490.328,E2 -490.328} C_VEL
LIN {X 0,Y 608.444,Z 274.689,A -85,B 0,C 180,E1 -492.96,E2 -492.96} C_VEL
LIN {X 0,Y 608.45,Z 274.688,A -85,B 0,C 180,E1 -495.736,E2 -495.736} C_VEL
LIN {X 0,Y 608.459,Z 274.694,A -85,B 0,C 180,E1 -498.657,E2 -498.657} C_VEL
LIN {X 0,Y 608.459,Z 274.686,A -85,B 0,C 180,E1 -501.411,E2 -501.411} C_VEL
LIN {X 0,Y 608.472,Z 274.685,A -85,B 0,C 180,E1 -503.95,E2 -503.95} C_VEL
LIN {X 0,Y 608.466,Z 274.69,A -85,B 0,C 180,E1 -506.329,E2 -506.329} C_VEL
LIN {X 0,Y 608.47,Z 274.696,A -85,B 0,C 180,E1 -508.726,E2 -508.726} C_VEL
LIN {X 0,Y 608.452,Z 274.689,A -85,B 0,C 180,E1 -511.381,E2 -511.381} C_VEL
LIN {X 0,Y 608.438,Z 274.688,A -85,B 0,C 180,E1 -513.964,E2 -513.964} C_VEL
LIN {X 0,Y 608.46,Z 274.686,A -85,B 0,C 180,E1 -516.155,E2 -516.155} C_VEL
LIN {X 0,Y 608.447,Z 274.698,A -85,B 0,C 180,E1 -519.018,E2 -519.018} C_VEL
LIN {X 0,Y 608.429,Z 274.69,A -85,B 0,C 180,E1 -521.827,E2 -521.827} C_VEL
LIN {X 0,Y 608.467,Z 274.687,A -85,B 0,C 180,E1 -524.594,E2 -524.594} C_VEL
LIN {X 0,Y 608.463,Z 274.694,A -85,B 0,C 180,E1 -527.323,E2 -527.323} C_VEL
LIN {X 0,Y 608.428,Z 274.69,A -85,B 0,C 180,E1 -530.022,E2 -530.022} C_VEL
LIN {X 0,Y 608.474,Z 274.686,A -85,B 0,C 180,E1 -532.701,E2 -532.701} C_VEL
LIN {X 0,Y 608.463,Z 274.697,A -85,B 0,C 180,E1 -535.362,E2 -535.362} C_VEL
LIN {X 0,Y 608.419,Z 274.693,A -85,B 0,C 180,E1 -538.014,E2 -538.014} C_VEL
LIN {X 0,Y 608.441,Z 274.691,A -85,B 0,C 180,E1 -540,E2 -540} C_VEL
LIN {X 0,Y 608.445,Z 274.687,A -85,B 0,C 180,E1 -542.648,E2 -542.648} C_VEL
LIN {X 0,Y 608.468,Z 274.69,A -85,B 0,C 180,E1 -545.302,E2 -545.302} C_VEL
LIN {X 0,Y 608.46,Z 274.692,A -85,B 0,C 180,E1 -547.967,E2 -547.967} C_VEL
LIN {X 0,Y 608.455,Z 274.69,A -85,B 0,C 180,E1 -549.437,E2 -549.437} C_VEL
LIN {X 0,Y 607.768,Z 274.779,A -85,B 0,C 180,E1 -549.989,E2 -549.989} C_VEL
LIN {X 0,Y 604.913,Z 275.134,A -85,B 0,C 180,E1 -550.886,E2 -550.886} C_VEL
LIN {X 0,Y 602.509,Z 275.435,A -85,B 0,C 180,E1 -551.607,E2 -551.607} C_VEL
LIN {X 0,Y 601.472,Z 275.561,A -85,B 0,C 180,E1 -552.164,E2 -552.164} C_VEL
LIN {X 0,Y 601.384,Z 275.569,A -85,B 0,C 180,E1 -552.352,E2 -552.352} C_VEL
LIN {X 0,Y 601.379,Z 275.568,A -85,B 0,C 180,E1 -554.898,E2 -554.898} C_VEL
LIN {X 0,Y 601.381,Z 275.575,A -85,B 0,C 180,E1 -557.689,E2 -557.689} C_VEL
LIN {X 0,Y 601.395,Z 275.568,A -85,B 0,C 180,E1 -560.523,E2 -560.523} C_VEL
LIN {X 0,Y 601.377,Z 275.569,A -85,B 0,C 180,E1 -563.412,E2 -563.412} C_VEL
LIN {X 0,Y 601.396,Z 275.572,A -85,B 0,C 180,E1 -565.867,E2 -565.867} C_VEL
LIN {X 0,Y 601.378,Z 275.57,A -85,B 0,C 180,E1 -568.781,E2 -568.781} C_VEL
LIN {X 0,Y 601.397,Z 275.566,A -85,B 0,C 180,E1 -571.453,E2 -571.453} C_VEL
LIN {X 0,Y 601.404,Z 275.573,A -85,B 0,C 180,E1 -574.12,E2 -574.12} C_VEL
LIN {X 0,Y 601.368,Z 275.576,A -85,B 0,C 180,E1 -576.586,E2 -576.586} C_VEL
LIN {X 0,Y 601.364,Z 275.57,A -85,B 0,C 180,E1 -579.13,E2 -579.13} C_VEL
LIN {X 0,Y 601.374,Z 275.569,A -85,B 0,C 180,E1 -581.77,E2 -581.77} C_VEL
LIN {X 0,Y 601.394,Z 275.577,A -85,B 0,C 180,E1 -584.533,E2 -584.533} C_VEL
LIN {X 0,Y 601.34,Z 275.573,A -85,B 0,C 180,E1 -587.324,E2 -587.324} C_VEL
LIN {X 0,Y 601.338,Z 275.573,A -85,B 0,C 180,E1 -589.436,E2 -589.436} C_VEL
LIN {X 0,Y 601.329,Z 275.574,A -85,B 0,C 180,E1 -591.726,E2 -591.726} C_VEL
LIN {X 0,Y 601.338,Z 275.575,A -85,B 0,C 180,E1 -594.242,E2 -594.242} C_VEL
LIN {X 0,Y 601.381,Z 275.571,A -85,B 0,C 180,E1 -597.291,E2 -597.291} C_VEL
LIN {X 0,Y 601.343,Z 275.572,A -85,B 0,C 180,E1 -599.866,E2 -599.866} C_VEL
LIN {X 0,Y 601.346,Z 275.572,A -85,B 0,C 180,E1 -602.129,E2 -602.129} C_VEL
LIN {X 0,Y 601.355,Z 275.572,A -85,B 0,C 180,E1 -604.378,E2 -604.378} C_VEL
LIN {X 0,Y 601.404,Z 275.572,A -85,B 0,C 180,E1 -607.316,E2 -607.316} C_VEL
LIN {X 0,Y 601.417,Z 275.568,A -85,B 0,C 180,E1 -609.477,E2 -609.477} C_VEL
LIN {X 0,Y 601.387,Z 275.571,A -85,B 0,C 180,E1 -611.606,E2 -611.606} C_VEL
LIN {X 0,Y 601.418,Z 275.566,A -85,B 0,C 180,E1 -613.711,E2 -613.711} C_VEL
LIN {X 0,Y 601.375,Z 275.568,A -85,B 0,C 180,E1 -616.482,E2 -616.482} C_VEL
LIN {X 0,Y 601.399,Z 275.574,A -85,B 0,C 180,E1 -619.222,E2 -619.222} C_VEL
LIN {X 0,Y 601.4,Z 275.568,A -85,B 0,C 180,E1 -621.937,E2 -621.937} C_VEL
LIN {X 0,Y 601.392,Z 275.569,A -85,B 0,C 180,E1 -623.961,E2 -623.961} C_VEL
LIN {X 0,Y 601.394,Z 275.569,A -85,B 0,C 180,E1 -625.977,E2 -625.977} C_VEL
LIN {X 0,Y 601.425,Z 275.566,A -85,B 0,C 180,E1 -627.989,E2 -627.989} C_VEL
LIN {X 0,Y 601.372,Z 275.568,A -85,B 0,C 180,E1 -630.667,E2 -630.667} C_VEL
LIN {X 0,Y 601.407,Z 275.564,A -85,B 0,C 180,E1 -632.677,E2 -632.677} C_VEL
LIN {X 0,Y 601.401,Z 275.569,A -85,B 0,C 180,E1 -635.362,E2 -635.362} C_VEL
LIN {X 0,Y 601.438,Z 275.568,A -85,B 0,C 180,E1 -638.058,E2 -638.058} C_VEL
LIN {X 0,Y 601.388,Z 275.567,A -85,B 0,C 180,E1 -640.774,E2 -640.774} C_VEL
LIN {X 0,Y 601.385,Z 275.657,A -85,B 0,C 180,E1 -643.255,E2 -643.255} C_VEL
LIN {X 0,Y 601.427,Z 287.091,A -85,B 0,C 180,E1 -645.24,E2 -645.24} C_VEL
LIN {X 0,Y 601.419,Z 303.407,A -85,B 0,C 180,E1 -648.036,E2 -648.036} C_VEL
LIN {X 0,Y 601.442,Z 308.522,A -85,B 0,C 180,E1 -648.89,E2 -648.89} C_VEL
LIN {X 0,Y 601.654,Z 322.659,A -85,B 0,C 180,E1 -649.065,E2 -649.065} C_VEL
LIN {X 0,Y 601.58,Z 414.622,A -85,B 0,C 180,E1 -650.178,E2 -650.178} C_VEL
LIN {X 0,Y 601.56,Z 427.722,A -85,B 0,C 180,E1 -650.469,E2 -650.469} C_VEL
LIN {X 0,Y 601.559,Z 440.456,A -85,B 0,C 180,E1 -650.892,E2 -650.892} C_VEL
LIN {X 0,Y 601.5,Z 452.071,A -85,B 0,C 180,E1 -651.412,E2 -651.412} C_VEL
LIN {X 0,Y 601.461,Z 463.026,A -85,B 0,C 180,E1 -652.043,E2 -652.043} C_VEL
LIN {X 0,Y 601.443,Z 474.287,A -85,B 0,C 180,E1 -652.859,E2 -652.859} C_VEL
LIN {X 0,Y 601.423,Z 482.442,A -85,B 0,C 180,E1 -653.589,E2 -653.589} C_VEL
LIN {X 0,Y 601.422,Z 491.407,A -85,B 0,C 180,E1 -654.545,E2 -654.545} C_VEL
LIN {X 0,Y 601.364,Z 499.377,A -85,B 0,C 180,E1 -655.616,E2 -655.616} C_VEL
LIN {X 0,Y 601.353,Z 505.98,A -85,B 0,C 180,E1 -656.736,E2 -656.736} C_VEL
LIN {X 0,Y 601.348,Z 511.096,A -85,B 0,C 180,E1 -657.866,E2 -657.866} C_VEL
LIN {X 0,Y 601.341,Z 514.198,A -85,B 0,C 180,E1 -658.772,E2 -658.772} C_VEL
LIN {X 0,Y 601.341,Z 515.875,A -85,B 0,C 180,E1 -659.393,E2 -659.393} C_VEL
LIN {X 0,Y 601.333,Z 517.413,A -85,B 0,C 180,E1 -660.164,E2 -660.164} C_VEL
LIN {X 0,Y 601.338,Z 518.83,A -85,B 0,C 180,E1 -661.441,E2 -661.441} C_VEL
LIN {X 0,Y 601.326,Z 518.794,A -85,B 0,C 180,E1 -662.701,E2 -662.701} C_VEL
LIN {X 0,Y 601.32,Z 517.423,A -85,B 0,C 180,E1 -663.919,E2 -663.919} C_VEL
LIN {X 0,Y 601.321,Z 514.816,A -85,B 0,C 180,E1 -665.101,E2 -665.101} C_VEL
LIN {X 0,Y 601.346,Z 510.986,A -85,B 0,C 180,E1 -666.253,E2 -666.253} C_VEL
LIN {X 0,Y 601.36,Z 505.631,A -85,B 0,C 180,E1 -667.419,E2 -667.419} C_VEL
LIN {X 0,Y 601.366,Z 498.596,A -85,B 0,C 180,E1 -668.591,E2 -668.591} C_VEL
LIN {X 0,Y 601.394,Z 491.532,A -85,B 0,C 180,E1 -669.53,E2 -669.53} C_VEL
LIN {X 0,Y 601.408,Z 483.301,A -85,B 0,C 180,E1 -670.416,E2 -670.416} C_VEL
LIN {X 0,Y 601.441,Z 474.687,A -85,B 0,C 180,E1 -671.199,E2 -671.199} C_VEL
LIN {X 0,Y 601.456,Z 464.033,A -85,B 0,C 180,E1 -671.981,E2 -671.981} C_VEL
LIN {X 0,Y 601.51,Z 452.522,A -85,B 0,C 180,E1 -672.655,E2 -672.655} C_VEL
LIN {X 0,Y 601.564,Z 441.352,A -85,B 0,C 180,E1 -673.164,E2 -673.164} C_VEL
LIN {X 0,Y 601.597,Z 428.236,A -85,B 0,C 180,E1 -673.606,E2 -673.606} C_VEL
LIN {X 0,Y 601.609,Z 415.568,A -85,B 0,C 180,E1 -673.894,E2 -673.894} C_VEL
LIN {X 0,Y 601.547,Z 309.467,A -85,B 0,C 180,E1 -675.186,E2 -675.186} C_VEL
LIN {X 0,Y 601.427,Z 308.366,A -85,B 0,C 180,E1 -675.211,E2 -675.211} C_VEL
LIN {X 0,Y 601.471,Z 290.631,A -85,B 0,C 180,E1 -678.239,E2 -678.239} C_VEL
LIN {X 0,Y 601.424,Z 275.726,A -85,B 0,C 180,E1 -680.821,E2 -680.821} C_VEL
LIN {X 0,Y 601.41,Z 275.568,A -85,B 0,C 180,E1 -683.729,E2 -683.729} C_VEL
LIN {X 0,Y 601.402,Z 275.569,A -85,B 0,C 180,E1 -686.685,E2 -686.685} C_VEL
LIN {X 0,Y 601.39,Z 275.567,A -85,B 0,C 180,E1 -689.056,E2 -689.056} C_VEL
LIN {X 0,Y 601.383,Z 275.568,A -85,B 0,C 180,E1 -691.37,E2 -691.37} C_VEL
LIN {X 0,Y 601.403,Z 275.571,A -85,B 0,C 180,E1 -694.121,E2 -694.121} C_VEL
LIN {X 0,Y 601.388,Z 275.575,A -85,B 0,C 180,E1 -696.588,E2 -696.588} C_VEL
LIN {X 0,Y 601.371,Z 275.569,A -85,B 0,C 180,E1 -699.476,E2 -699.476} C_VEL
LIN {X 0,Y 601.363,Z 275.577,A -85,B 0,C 180,E1 -702.311,E2 -702.311} C_VEL
LIN {X 0,Y 601.378,Z 275.571,A -85,B 0,C 180,E1 -705.102,E2 -705.102} C_VEL
LIN {X 0,Y 601.358,Z 275.571,A -85,B 0,C 180,E1 -707.856,E2 -707.856} C_VEL
LIN {X 0,Y 601.369,Z 275.569,A -85,B 0,C 180,E1 -709.904,E2 -709.904} C_VEL
LIN {X 0,Y 601.41,Z 275.573,A -85,B 0,C 180,E1 -712.614,E2 -712.614} C_VEL
LIN {X 0,Y 601.368,Z 275.572,A -85,B 0,C 180,E1 -715.308,E2 -715.308} C_VEL
LIN {X 0,Y 601.393,Z 275.569,A -85,B 0,C 180,E1 -717.321,E2 -717.321} C_VEL
LIN {X 0,Y 601.374,Z 275.568,A -85,B 0,C 180,E1 -720,E2 -720} C_VEL
LIN {X 0,Y 601.409,Z 275.571,A -85,B 0,C 180,E1 -722.679,E2 -722.679} C_VEL
LIN {X 0,Y 601.41,Z 275.568,A -85,B 0,C 180,E1 -725.364,E2 -725.364} C_VEL
LIN {X 0,Y 601.387,Z 275.566,A -85,B 0,C 180,E1 -728.062,E2 -728.062} C_VEL
LIN {X 0,Y 601.433,Z 275.572,A -85,B 0,C 180,E1 -731.047,E2 -731.047} C_VEL
LIN {X 0,Y 601.397,Z 275.57,A -85,B 0,C 180,E1 -733.516,E2 -733.516} C_VEL
LIN {X 0,Y 601.403,Z 275.565,A -85,B 0,C 180,E1 -736.288,E2 -736.288} C_VEL
LIN {X 0,Y 601.394,Z 275.575,A -85,B 0,C 180,E1 -739.1,E2 -739.1} C_VEL
LIN {X 0,Y 601.388,Z 275.568,A -85,B 0,C 180,E1 -741.96,E2 -741.96} C_VEL
LIN {X 0,Y 601.406,Z 275.564,A -85,B 0,C 180,E1 -744.3,E2 -744.3} C_VEL
LIN {X 0,Y 601.424,Z 275.569,A -85,B 0,C 180,E1 -747.113,E2 -747.113} C_VEL
LIN {X 0,Y 601.409,Z 275.565,A -85,B 0,C 180,E1 -750.156,E2 -750.156} C_VEL
LIN {X 0,Y 601.395,Z 275.566,A -85,B 0,C 180,E1 -752.722,E2 -752.722} C_VEL
LIN {X 0,Y 601.392,Z 275.57,A -85,B 0,C 180,E1 -755.121,E2 -755.121} C_VEL
LIN {X 0,Y 601.406,Z 275.573,A -85,B 0,C 180,E1 -757.421,E2 -757.421} C_VEL
LIN {X 0,Y 601.413,Z 275.568,A -85,B 0,C 180,E1 -759.995,E2 -759.995} C_VEL
LIN {X 0,Y 601.418,Z 275.563,A -85,B 0,C 180,E1 -762.67,E2 -762.67} C_VEL
LIN {X 0,Y 601.394,Z 275.573,A -85,B 0,C 180,E1 -765.486,E2 -765.486} C_VEL
LIN {X 0,Y 601.416,Z 275.565,A -85,B 0,C 180,E1 -768.408,E2 -768.408} C_VEL
LIN {X 0,Y 601.42,Z 275.563,A -85,B 0,C 180,E1 -770.88,E2 -770.88} C_VEL
LIN {X 0,Y 601.425,Z 275.571,A -85,B 0,C 180,E1 -773.737,E2 -773.737} C_VEL
LIN {X 0,Y 601.419,Z 275.564,A -85,B 0,C 180,E1 -776.691,E2 -776.691} C_VEL
LIN {X 0,Y 601.421,Z 275.563,A -85,B 0,C 180,E1 -779.063,E2 -779.063} C_VEL
LIN {X 0,Y 601.424,Z 275.564,A -85,B 0,C 180,E1 -781.377,E2 -781.377} C_VEL
LIN {X 0,Y 601.397,Z 275.57,A -85,B 0,C 180,E1 -783.64,E2 -783.64} C_VEL
LIN {X 0,Y 601.416,Z 275.57,A -85,B 0,C 180,E1 -786.594,E2 -786.594} C_VEL
LIN {X 0,Y 601.438,Z 275.608,A -85,B 0,C 180,E1 -787.141,E2 -787.141} C_VEL
LIN {X 0,Y 601.671,Z 282.079,A -85,B 0,C 180,E1 -788.055,E2 -788.055} C_VEL
LIN {X 0,Y 601.596,Z 302.79,A -85,B 0,C 180,E1 -790.911,E2 -790.911} C_VEL
LIN {X 0,Y 601.524,Z 323.5,A -85,B 0,C 180,E1 -793.719,E2 -793.719} C_VEL
LIN {X 0,Y 601.468,Z 344.21,A -85,B 0,C 180,E1 -796.488,E2 -796.488} C_VEL
LIN {X 0,Y 601.437,Z 346.718,A -85,B 0,C 180,E1 -796.821,E2 -796.821} C_VEL
LIN {X 0,Y 601.64,Z 358.137,A -85,B 0,C 180,E1 -796.965,E2 -796.965} C_VEL
LIN {X 0,Y 601.592,Z 455.11,A -85,B 0,C 180,E1 -798.142,E2 -798.142} C_VEL
LIN {X 0,Y 601.554,Z 468.325,A -85,B 0,C 180,E1 -798.44,E2 -798.44} C_VEL
LIN {X 0,Y 601.537,Z 480.696,A -85,B 0,C 180,E1 -798.855,E2 -798.855} C_VEL
LIN {X 0,Y 601.52,Z 492.689,A -85,B 0,C 180,E1 -799.399,E2 -799.399} C_VEL
LIN {X 0,Y 601.472,Z 504.242,A -85,B 0,C 180,E1 -800.078,E2 -800.078} C_VEL
LIN {X 0,Y 601.444,Z 514.631,A -85,B 0,C 180,E1 -800.842,E2 -800.842} C_VEL
LIN {X 0,Y 601.428,Z 523.043,A -85,B 0,C 180,E1 -801.604,E2 -801.604} C_VEL
LIN {X 0,Y 601.416,Z 530.984,A -85,B 0,C 180,E1 -802.448,E2 -802.448} C_VEL
LIN {X 0,Y 601.363,Z 538.262,A -85,B 0,C 180,E1 -803.404,E2 -803.404} C_VEL
LIN {X 0,Y 601.371,Z 543.88,A -85,B 0,C 180,E1 -804.302,E2 -804.302} C_VEL
LIN {X 0,Y 601.336,Z 548.961,A -85,B 0,C 180,E1 -805.31,E2 -805.31} C_VEL
LIN {X 0,Y 601.367,Z 552.904,A -85,B 0,C 180,E1 -806.317,E2 -806.317} C_VEL
LIN {X 0,Y 601.325,Z 555.815,A -85,B 0,C 180,E1 -807.323,E2 -807.323} C_VEL
LIN {X 0,Y 601.341,Z 557.205,A -85,B 0,C 180,E1 -807.993,E2 -807.993} C_VEL
LIN {X 0,Y 601.339,Z 558.785,A -85,B 0,C 180,E1 -809.333,E2 -809.333} C_VEL
LIN {X 0,Y 601.335,Z 559,A -85,B 0,C 180,E1 -810.002,E2 -810.002} C_VEL
LIN {X 0,Y 601.347,Z 558.182,A -85,B 0,C 180,E1 -811.341,E2 -811.341} C_VEL
LIN {X 0,Y 601.341,Z 557.199,A -85,B 0,C 180,E1 -812.011,E2 -812.011} C_VEL
LIN {X 0,Y 601.325,Z 555.804,A -85,B 0,C 180,E1 -812.682,E2 -812.682} C_VEL
LIN {X 0,Y 601.367,Z 552.89,A -85,B 0,C 180,E1 -813.687,E2 -813.687} C_VEL
LIN {X 0,Y 601.336,Z 548.942,A -85,B 0,C 180,E1 -814.695,E2 -814.695} C_VEL
LIN {X 0,Y 601.372,Z 542.866,A -85,B 0,C 180,E1 -815.871,E2 -815.871} C_VEL
LIN {X 0,Y 601.383,Z 536.223,A -85,B 0,C 180,E1 -816.881,E2 -816.881} C_VEL
LIN {X 0,Y 601.401,Z 527.975,A -85,B 0,C 180,E1 -817.894,E2 -817.894} C_VEL
LIN {X 0,Y 601.435,Z 517.581,A -85,B 0,C 180,E1 -818.909,E2 -818.909} C_VEL
LIN {X 0,Y 601.46,Z 506.725,A -85,B 0,C 180,E1 -819.756,E2 -819.756} C_VEL
LIN {X 0,Y 601.494,Z 495.748,A -85,B 0,C 180,E1 -820.436,E2 -820.436} C_VEL
LIN {X 0,Y 601.55,Z 483.669,A -85,B 0,C 180,E1 -821.022,E2 -821.022} C_VEL
LIN {X 0,Y 601.531,Z 471.834,A -85,B 0,C 180,E1 -821.458,E2 -821.458} C_VEL
LIN {X 0,Y 601.578,Z 459.436,A -85,B 0,C 180,E1 -821.777,E2 -821.777} C_VEL
LIN {X 0,Y 601.608,Z 443.616,A -85,B 0,C 180,E1 -822.012,E2 -822.012} C_VEL
LIN {X 0,Y 601.479,Z 347.033,A -85,B 0,C 180,E1 -823.172,E2 -823.172} C_VEL
LIN {X 0,Y 601.468,Z 344.176,A -85,B 0,C 180,E1 -823.516,E2 -823.516} C_VEL
LIN {X 0,Y 601.52,Z 323.466,A -85,B 0,C 180,E1 -826.286,E2 -826.286} C_VEL
LIN {X 0,Y 601.604,Z 302.756,A -85,B 0,C 180,E1 -829.094,E2 -829.094} C_VEL
LIN {X 0,Y 601.697,Z 280.772,A -85,B 0,C 180,E1 -832.127,E2 -832.127} C_VEL
LIN {X 0,Y 601.422,Z 275.574,A -85,B 0,C 180,E1 -832.865,E2 -832.865} C_VEL
LIN {X 0,Y 601.399,Z 275.566,A -85,B 0,C 180,E1 -834.879,E2 -834.879} C_VEL
LIN {X 0,Y 601.414,Z 275.565,A -85,B 0,C 180,E1 -837.362,E2 -837.362} C_VEL
LIN {X 0,Y 601.431,Z 275.571,A -85,B 0,C 180,E1 -840.164,E2 -840.164} C_VEL
LIN {X 0,Y 601.418,Z 275.565,A -85,B 0,C 180,E1 -842.714,E2 -842.714} C_VEL
LIN {X 0,Y 601.391,Z 275.566,A -85,B 0,C 180,E1 -845.111,E2 -845.111} C_VEL
LIN {X 0,Y 601.436,Z 275.561,A -85,B 0,C 180,E1 -847.419,E2 -847.419} C_VEL
LIN {X 0,Y 601.4,Z 275.571,A -85,B 0,C 180,E1 -849.995,E2 -849.995} C_VEL
LIN {X 0,Y 601.411,Z 275.569,A -85,B 0,C 180,E1 -852.67,E2 -852.67} C_VEL
LIN {X 0,Y 601.395,Z 275.566,A -85,B 0,C 180,E1 -855.479,E2 -855.479} C_VEL
LIN {X 0,Y 601.422,Z 275.572,A -85,B 0,C 180,E1 -858.406,E2 -858.406} C_VEL
LIN {X 0,Y 601.426,Z 275.567,A -85,B 0,C 180,E1 -860.874,E2 -860.874} C_VEL
LIN {X 0,Y 601.436,Z 275.561,A -85,B 0,C 180,E1 -863.733,E2 -863.733} C_VEL
LIN {X 0,Y 601.425,Z 275.574,A -85,B 0,C 180,E1 -866.686,E2 -866.686} C_VEL
LIN {X 0,Y 601.422,Z 275.568,A -85,B 0,C 180,E1 -869.058,E2 -869.058} C_VEL
LIN {X 0,Y 601.413,Z 275.566,A -85,B 0,C 180,E1 -871.372,E2 -871.372} C_VEL
LIN {X 0,Y 601.394,Z 275.566,A -85,B 0,C 180,E1 -873.636,E2 -873.636} C_VEL
LIN {X 0,Y 601.414,Z 275.568,A -85,B 0,C 180,E1 -876.589,E2 -876.589} C_VEL
LIN {X 0,Y 601.411,Z 275.567,A -85,B 0,C 180,E1 -879.477,E2 -879.477} C_VEL
LIN {X 0,Y 601.387,Z 275.567,A -85,B 0,C 180,E1 -882.311,E2 -882.311} C_VEL
LIN {X 0,Y 601.419,Z 275.574,A -85,B 0,C 180,E1 -885.103,E2 -885.103} C_VEL
LIN {X 0,Y 601.397,Z 275.567,A -85,B 0,C 180,E1 -887.857,E2 -887.857} C_VEL
LIN {X 0,Y 601.413,Z 275.565,A -85,B 0,C 180,E1 -890.584,E2 -890.584} C_VEL
LIN {X 0,Y 601.439,Z 275.572,A -85,B 0,C 180,E1 -893.324,E2 -893.324} C_VEL
LIN {X 0,Y 601.375,Z 275.57,A -85,B 0,C 180,E1 -895.979,E2 -895.979} C_VEL
LIN {X 0,Y 601.392,Z 275.568,A -85,B 0,C 180,E1 -897.991,E2 -897.991} C_VEL
LIN {X 0,Y 601.411,Z 275.566,A -85,B 0,C 180,E1 -900,E2 -900} C_VEL
LIN {X 0,Y 601.414,Z 275.563,A -85,B 0,C 180,E1 -902.679,E2 -902.679} C_VEL
LIN {X 0,Y 601.428,Z 275.568,A -85,B 0,C 180,E1 -905.364,E2 -905.364} C_VEL
LIN {X 0,Y 601.42,Z 275.567,A -85,B 0,C 180,E1 -908.061,E2 -908.061} C_VEL
LIN {X 0,Y 601.379,Z 275.568,A -85,B 0,C 180,E1 -910.777,E2 -910.777} C_VEL
LIN {X 0,Y 601.384,Z 275.569,A -85,B 0,C 180,E1 -912.352,E2 -912.352} C_VEL
LIN {X 0,Y 600.708,Z 275.654,A -85,B 0,C 180,E1 -912.912,E2 -912.912} C_VEL
LIN {X 0,Y 597.85,Z 276.019,A -85,B 0,C 180,E1 -913.819,E2 -913.819} C_VEL
LIN {X 0,Y 595.442,Z 276.312,A -85,B 0,C 180,E1 -914.549,E2 -914.549} C_VEL
LIN {X 0,Y 594.411,Z 276.437,A -85,B 0,C 180,E1 -915.113,E2 -915.113} C_VEL
LIN {X 0,Y 594.328,Z 276.448,A -85,B 0,C 180,E1 -915.304,E2 -915.304} C_VEL
LIN {X 0,Y 594.358,Z 276.454,A -85,B 0,C 180,E1 -917.905,E2 -917.905} C_VEL
LIN {X 0,Y 594.344,Z 276.444,A -85,B 0,C 180,E1 -920.912,E2 -920.912} C_VEL
LIN {X 0,Y 594.357,Z 276.447,A -85,B 0,C 180,E1 -923.706,E2 -923.706} C_VEL
LIN {X 0,Y 594.347,Z 276.453,A -85,B 0,C 180,E1 -926.018,E2 -926.018} C_VEL
LIN {X 0,Y 594.326,Z 276.447,A -85,B 0,C 180,E1 -929.002,E2 -929.002} C_VEL
LIN {X 0,Y 594.359,Z 276.444,A -85,B 0,C 180,E1 -931.642,E2 -931.642} C_VEL
LIN {X 0,Y 594.357,Z 276.451,A -85,B 0,C 180,E1 -934.137,E2 -934.137} C_VEL
LIN {X 0,Y 594.313,Z 276.449,A -85,B 0,C 180,E1 -937.092,E2 -937.092} C_VEL
LIN {X 0,Y 594.329,Z 276.447,A -85,B 0,C 180,E1 -939.77,E2 -939.77} C_VEL
LIN {X 0,Y 594.337,Z 276.454,A -85,B 0,C 180,E1 -942.378,E2 -942.378} C_VEL
LIN {X 0,Y 594.309,Z 276.45,A -85,B 0,C 180,E1 -945.197,E2 -945.197} C_VEL
LIN {X 0,Y 594.309,Z 276.448,A -85,B 0,C 180,E1 -947.62,E2 -947.62} C_VEL
LIN {X 0,Y 594.337,Z 276.45,A -85,B 0,C 180,E1 -950.317,E2 -950.317} C_VEL
LIN {X 0,Y 594.326,Z 276.454,A -85,B 0,C 180,E1 -952.909,E2 -952.909} C_VEL
LIN {X 0,Y 594.291,Z 276.451,A -85,B 0,C 180,E1 -955.875,E2 -955.875} C_VEL
LIN {X 0,Y 594.339,Z 276.451,A -85,B 0,C 180,E1 -958.648,E2 -958.648} C_VEL
LIN {X 0,Y 594.342,Z 276.454,A -85,B 0,C 180,E1 -961.05,E2 -961.05} C_VEL
LIN {X 0,Y 594.353,Z 276.449,A -85,B 0,C 180,E1 -963.298,E2 -963.298} C_VEL
LIN {X 0,Y 594.33,Z 276.446,A -85,B 0,C 180,E1 -966.293,E2 -966.293} C_VEL
LIN {X 0,Y 594.4,Z 276.447,A -85,B 0,C 180,E1 -969.223,E2 -969.223} C_VEL
LIN {X 0,Y 594.32,Z 276.447,A -85,B 0,C 180,E1 -972.093,E2 -972.093} C_VEL
LIN {X 0,Y 594.331,Z 276.446,A -85,B 0,C 180,E1 -974.217,E2 -974.217} C_VEL
LIN {X 0,Y 594.346,Z 276.449,A -85,B 0,C 180,E1 -977.015,E2 -977.015} C_VEL
LIN {X 0,Y 594.34,Z 276.449,A -85,B 0,C 180,E1 -979.782,E2 -979.782} C_VEL
LIN {X 0,Y 594.355,Z 276.447,A -85,B 0,C 180,E1 -981.841,E2 -981.841} C_VEL
LIN {X 0,Y 594.354,Z 276.443,A -85,B 0,C 180,E1 -984.57,E2 -984.57} C_VEL
LIN {X 0,Y 594.392,Z 276.444,A -85,B 0,C 180,E1 -987.287,E2 -987.287} C_VEL
LIN {X 0,Y 594.414,Z 276.44,A -85,B 0,C 180,E1 -989.998,E2 -989.998} C_VEL
LIN {X 0,Y 594.375,Z 276.44,A -85,B 0,C 180,E1 -992.709,E2 -992.709} C_VEL
LIN {X 0,Y 594.369,Z 276.446,A -85,B 0,C 180,E1 -995.425,E2 -995.425} C_VEL
LIN {X 0,Y 594.381,Z 276.445,A -85,B 0,C 180,E1 -998.154,E2 -998.154} C_VEL
LIN {X 0,Y 594.33,Z 276.447,A -85,B 0,C 180,E1 -1001.043,E2 -1001.043} C_VEL
LIN {X 0,Y 594.368,Z 276.632,A -85,B 0,C 180,E1 -1003.197,E2 -1003.197} C_VEL
LIN {X 0,Y 594.414,Z 288.31,A -85,B 0,C 180,E1 -1005.249,E2 -1005.249} C_VEL
LIN {X 0,Y 594.395,Z 303.6,A -85,B 0,C 180,E1 -1007.9,E2 -1007.9} C_VEL
LIN {X 0,Y 594.384,Z 308.401,A -85,B 0,C 180,E1 -1008.726,E2 -1008.726} C_VEL
LIN {X 0,Y 594.771,Z 314.398,A -85,B 0,C 180,E1 -1008.812,E2 -1008.812} C_VEL
LIN {X 0,Y 594.634,Z 414.814,A -85,B 0,C 180,E1 -1010.041,E2 -1010.041} C_VEL
LIN {X 0,Y 594.605,Z 427.847,A -85,B 0,C 180,E1 -1010.335,E2 -1010.335} C_VEL
LIN {X 0,Y 594.589,Z 440.607,A -85,B 0,C 180,E1 -1010.765,E2 -1010.765} C_VEL
LIN {X 0,Y 594.514,Z 451.541,A -85,B 0,C 180,E1 -1011.259,E2 -1011.259} C_VEL
LIN {X 0,Y 594.432,Z 462.09,A -85,B 0,C 180,E1 -1011.861,E2 -1011.861} C_VEL
LIN {X 0,Y 594.427,Z 473.228,A -85,B 0,C 180,E1 -1012.664,E2 -1012.664} C_VEL
LIN {X 0,Y 594.387,Z 482.729,A -85,B 0,C 180,E1 -1013.515,E2 -1013.515} C_VEL
LIN {X 0,Y 594.338,Z 491.321,A -85,B 0,C 180,E1 -1014.444,E2 -1014.444} C_VEL
LIN {X 0,Y 594.305,Z 499.558,A -85,B 0,C 180,E1 -1015.567,E2 -1015.567} C_VEL
LIN {X 0,Y 594.282,Z 506.125,A -85,B 0,C 180,E1 -1016.7,E2 -1016.7} C_VEL
LIN {X 0,Y 594.257,Z 511.197,A -85,B 0,C 180,E1 -1017.844,E2 -1017.844} C_VEL
LIN {X 0,Y 594.245,Z 514.945,A -85,B 0,C 180,E1 -1019.001,E2 -1019.001} C_VEL
LIN {X 0,Y 594.23,Z 517.673,A -85,B 0,C 180,E1 -1020.302,E2 -1020.302} C_VEL
LIN {X 0,Y 594.232,Z 518.908,A -85,B 0,C 180,E1 -1021.619,E2 -1021.619} C_VEL
LIN {X 0,Y 594.234,Z 518.625,A -85,B 0,C 180,E1 -1022.954,E2 -1022.954} C_VEL
LIN {X 0,Y 594.239,Z 517.136,A -85,B 0,C 180,E1 -1024.118,E2 -1024.118} C_VEL
LIN {X 0,Y 594.226,Z 514.029,A -85,B 0,C 180,E1 -1025.412,E2 -1025.412} C_VEL
LIN {X 0,Y 594.269,Z 510.313,A -85,B 0,C 180,E1 -1026.468,E2 -1026.468} C_VEL
LIN {X 0,Y 594.26,Z 505.053,A -85,B 0,C 180,E1 -1027.592,E2 -1027.592} C_VEL
LIN {X 0,Y 594.296,Z 498.44,A -85,B 0,C 180,E1 -1028.693,E2 -1028.693} C_VEL
LIN {X 0,Y 594.327,Z 491.059,A -85,B 0,C 180,E1 -1029.678,E2 -1029.678} C_VEL
LIN {X 0,Y 594.37,Z 482.872,A -85,B 0,C 180,E1 -1030.561,E2 -1030.561} C_VEL
LIN {X 0,Y 594.404,Z 473.937,A -85,B 0,C 180,E1 -1031.369,E2 -1031.369} C_VEL
LIN {X 0,Y 594.452,Z 463.633,A -85,B 0,C 180,E1 -1032.126,E2 -1032.126} C_VEL
LIN {X 0,Y 594.511,Z 452.071,A -85,B 0,C 180,E1 -1032.805,E2 -1032.805} C_VEL
LIN {X 0,Y 594.597,Z 440.559,A -85,B 0,C 180,E1 -1033.327,E2 -1033.327} C_VEL
LIN {X 0,Y 594.634,Z 427.97,A -85,B 0,C 180,E1 -1033.751,E2 -1033.751} C_VEL
LIN {X 0,Y 594.645,Z 414.806,A -85,B 0,C 180,E1 -1034.049,E2 -1034.049} C_VEL
LIN {X 0,Y 594.608,Z 309.912,A -85,B 0,C 180,E1 -1035.337,E2 -1035.337} C_VEL
LIN {X 0,Y 594.391,Z 308.249,A -85,B 0,C 180,E1 -1035.39,E2 -1035.39} C_VEL
LIN {X 0,Y 594.449,Z 291.188,A -85,B 0,C 180,E1 -1038.338,E2 -1038.338} C_VEL
LIN {X 0,Y 594.448,Z 277.348,A -85,B 0,C 180,E1 -1040.764,E2 -1040.764} C_VEL
LIN {X 0,Y 594.354,Z 276.447,A -85,B 0,C 180,E1 -1040.975,E2 -1040.975} C_VEL
LIN {X 0,Y 594.362,Z 276.446,A -85,B 0,C 180,E1 -1043.756,E2 -1043.756} C_VEL
LIN {X 0,Y 594.357,Z 276.454,A -85,B 0,C 180,E1 -1046.237,E2 -1046.237} C_VEL
LIN {X 0,Y 594.35,Z 276.448,A -85,B 0,C 180,E1 -1048.648,E2 -1048.648} C_VEL
LIN {X 0,Y 594.342,Z 276.446,A -85,B 0,C 180,E1 -1051.038,E2 -1051.038} C_VEL
LIN {X 0,Y 594.359,Z 276.448,A -85,B 0,C 180,E1 -1054.055,E2 -1054.055} C_VEL
LIN {X 0,Y 594.356,Z 276.452,A -85,B 0,C 180,E1 -1056.294,E2 -1056.294} C_VEL
LIN {X 0,Y 594.344,Z 276.445,A -85,B 0,C 180,E1 -1059.222,E2 -1059.222} C_VEL
LIN {X 0,Y 594.336,Z 276.449,A -85,B 0,C 180,E1 -1062.094,E2 -1062.094} C_VEL
LIN {X 0,Y 594.326,Z 276.452,A -85,B 0,C 180,E1 -1064.921,E2 -1064.921} C_VEL
LIN {X 0,Y 594.332,Z 276.446,A -85,B 0,C 180,E1 -1067.71,E2 -1067.71} C_VEL
LIN {X 0,Y 594.33,Z 276.446,A -85,B 0,C 180,E1 -1069.783,E2 -1069.783} C_VEL
LIN {X 0,Y 594.369,Z 276.449,A -85,B 0,C 180,E1 -1072.526,E2 -1072.526} C_VEL
LIN {X 0,Y 594.341,Z 276.448,A -85,B 0,C 180,E1 -1075.252,E2 -1075.252} C_VEL
LIN {X 0,Y 594.328,Z 276.446,A -85,B 0,C 180,E1 -1077.967,E2 -1077.967} C_VEL
LIN {X 0,Y 594.39,Z 276.445,A -85,B 0,C 180,E1 -1080.677,E2 -1080.677} C_VEL
LIN {X 0,Y 594.356,Z 276.446,A -85,B 0,C 180,E1 -1083.389,E2 -1083.389} C_VEL
LIN {X 0,Y 594.312,Z 276.448,A -85,B 0,C 180,E1 -1086.11,E2 -1086.11} C_VEL
LIN {X 0,Y 594.364,Z 276.441,A -85,B 0,C 180,E1 -1088.157,E2 -1088.157} C_VEL
LIN {X 0,Y 594.403,Z 276.447,A -85,B 0,C 180,E1 -1091.111,E2 -1091.111} C_VEL
LIN {X 0,Y 594.333,Z 276.446,A -85,B 0,C 180,E1 -1094.177,E2 -1094.177} C_VEL
LIN {X 0,Y 594.347,Z 276.447,A -85,B 0,C 180,E1 -1096.725,E2 -1096.725} C_VEL
LIN {X 0,Y 594.339,Z 276.454,A -85,B 0,C 180,E1 -1099.335,E2 -1099.335} C_VEL
LIN {X 0,Y 594.349,Z 276.45,A -85,B 0,C 180,E1 -1101.504,E2 -1101.504} C_VEL
LIN {X 0,Y 594.366,Z 276.445,A -85,B 0,C 180,E1 -1103.705,E2 -1103.705} C_VEL
LIN {X 0,Y 594.357,Z 276.444,A -85,B 0,C 180,E1 -1106.701,E2 -1106.701} C_VEL
LIN {X 0,Y 594.377,Z 276.444,A -85,B 0,C 180,E1 -1108.999,E2 -1108.999} C_VEL
LIN {X 0,Y 594.362,Z 276.449,A -85,B 0,C 180,E1 -1111.651,E2 -1111.651} C_VEL
LIN {X 0,Y 594.367,Z 276.441,A -85,B 0,C 180,E1 -1114.581,E2 -1114.581} C_VEL
LIN {X 0,Y 594.355,Z 276.446,A -85,B 0,C 180,E1 -1117.089,E2 -1117.089} C_VEL
LIN {X 0,Y 594.368,Z 276.449,A -85,B 0,C 180,E1 -1119.782,E2 -1119.782} C_VEL
LIN {X 0,Y 594.37,Z 276.442,A -85,B 0,C 180,E1 -1122.375,E2 -1122.375} C_VEL
LIN {X 0,Y 594.331,Z 276.449,A -85,B 0,C 180,E1 -1125.195,E2 -1125.195} C_VEL
LIN {X 0,Y 594.368,Z 276.451,A -85,B 0,C 180,E1 -1127.631,E2 -1127.631} C_VEL
LIN {X 0,Y 594.378,Z 276.443,A -85,B 0,C 180,E1 -1130.326,E2 -1130.326} C_VEL
LIN {X 0,Y 594.37,Z 276.441,A -85,B 0,C 180,E1 -1132.918,E2 -1132.918} C_VEL
LIN {X 0,Y 594.372,Z 276.452,A -85,B 0,C 180,E1 -1135.863,E2 -1135.863} C_VEL
LIN {X 0,Y 594.376,Z 276.442,A -85,B 0,C 180,E1 -1138.655,E2 -1138.655} C_VEL
LIN {X 0,Y 594.373,Z 276.441,A -85,B 0,C 180,E1 -1141.044,E2 -1141.044} C_VEL
LIN {X 0,Y 594.379,Z 276.45,A -85,B 0,C 180,E1 -1143.979,E2 -1143.979} C_VEL
LIN {X 0,Y 594.37,Z 276.447,A -85,B 0,C 180,E1 -1146.853,E2 -1146.853} C_VEL
LIN {X 0,Y 594.415,Z 276.578,A -85,B 0,C 180,E1 -1146.993,E2 -1146.993} C_VEL
LIN {X 0,Y 594.77,Z 283.374,A -85,B 0,C 180,E1 -1147.969,E2 -1147.969} C_VEL
LIN {X 0,Y 594.632,Z 304.394,A -85,B 0,C 180,E1 -1150.901,E2 -1150.901} C_VEL
LIN {X 0,Y 594.513,Z 324.794,A -85,B 0,C 180,E1 -1153.698,E2 -1153.698} C_VEL
LIN {X 0,Y 594.438,Z 345.504,A -85,B 0,C 180,E1 -1156.5,E2 -1156.5} C_VEL
LIN {X 0,Y 594.433,Z 346.718,A -85,B 0,C 180,E1 -1156.663,E2 -1156.663} C_VEL
LIN {X 0,Y 594.763,Z 352.771,A -85,B 0,C 180,E1 -1156.747,E2 -1156.747} C_VEL
LIN {X 0,Y 594.643,Z 455.11,A -85,B 0,C 180,E1 -1158.002,E2 -1158.002} C_VEL
LIN {X 0,Y 594.617,Z 468.326,A -85,B 0,C 180,E1 -1158.304,E2 -1158.304} C_VEL
LIN {X 0,Y 594.557,Z 481.274,A -85,B 0,C 180,E1 -1158.745,E2 -1158.745} C_VEL
LIN {X 0,Y 594.532,Z 492.687,A -85,B 0,C 180,E1 -1159.273,E2 -1159.273} C_VEL
LIN {X 0,Y 594.459,Z 504.244,A -85,B 0,C 180,E1 -1159.96,E2 -1159.96} C_VEL
LIN {X 0,Y 594.413,Z 514.632,A -85,B 0,C 180,E1 -1160.732,E2 -1160.732} C_VEL
LIN {X 0,Y 594.365,Z 523.057,A -85,B 0,C 180,E1 -1161.503,E2 -1161.503} C_VEL
LIN {X 0,Y 594.346,Z 530.984,A -85,B 0,C 180,E1 -1162.358,E2 -1162.358} C_VEL
LIN {X 0,Y 594.278,Z 538.837,A -85,B 0,C 180,E1 -1163.412,E2 -1163.412} C_VEL
LIN {X 0,Y 594.289,Z 545.694,A -85,B 0,C 180,E1 -1164.574,E2 -1164.574} C_VEL
LIN {X 0,Y 594.27,Z 550.382,A -85,B 0,C 180,E1 -1165.594,E2 -1165.594} C_VEL
LIN {X 0,Y 594.267,Z 553.964,A -85,B 0,C 180,E1 -1166.612,E2 -1166.612} C_VEL
LIN {X 0,Y 594.226,Z 555.815,A -85,B 0,C 180,E1 -1167.291,E2 -1167.291} C_VEL
LIN {X 0,Y 594.24,Z 557.205,A -85,B 0,C 180,E1 -1167.969,E2 -1167.969} C_VEL
LIN {X 0,Y 594.239,Z 558.786,A -85,B 0,C 180,E1 -1169.325,E2 -1169.325} C_VEL
LIN {X 0,Y 594.236,Z 559,A -85,B 0,C 180,E1 -1170.002,E2 -1170.002} C_VEL
LIN {X 0,Y 594.247,Z 558.182,A -85,B 0,C 180,E1 -1171.357,E2 -1171.357} C_VEL
LIN {X 0,Y 594.24,Z 557.198,A -85,B 0,C 180,E1 -1172.035,E2 -1172.035} C_VEL
LIN {X 0,Y 594.226,Z 555.805,A -85,B 0,C 180,E1 -1172.714,E2 -1172.714} C_VEL
LIN {X 0,Y 594.289,Z 552.89,A -85,B 0,C 180,E1 -1173.731,E2 -1173.731} C_VEL
LIN {X 0,Y 594.241,Z 548.942,A -85,B 0,C 180,E1 -1174.751,E2 -1174.751} C_VEL
LIN {X 0,Y 594.304,Z 542.867,A -85,B 0,C 180,E1 -1175.941,E2 -1175.941} C_VEL
LIN {X 0,Y 594.309,Z 536.224,A -85,B 0,C 180,E1 -1176.964,E2 -1176.964} C_VEL
LIN {X 0,Y 594.36,Z 527.975,A -85,B 0,C 180,E1 -1177.988,E2 -1177.988} C_VEL
LIN {X 0,Y 594.405,Z 517.582,A -85,B 0,C 180,E1 -1179.015,E2 -1179.015} C_VEL
LIN {X 0,Y 594.448,Z 506.725,A -85,B 0,C 180,E1 -1179.872,E2 -1179.872} C_VEL
LIN {X 0,Y 594.506,Z 495.75,A -85,B 0,C 180,E1 -1180.56,E2 -1180.56} C_VEL
LIN {X 0,Y 594.567,Z 483.552,A -85,B 0,C 180,E1 -1181.159,E2 -1181.159} C_VEL
LIN {X 0,Y 594.576,Z 471.832,A -85,B 0,C 180,E1 -1181.594,E2 -1181.594} C_VEL
LIN {X 0,Y 594.634,Z 459.435,A -85,B 0,C 180,E1 -1181.917,E2 -1181.917} C_VEL
LIN {X 0,Y 594.69,Z 443.616,A -85,B 0,C 180,E1 -1182.153,E2 -1182.153} C_VEL
LIN {X 0,Y 594.623,Z 348.152,A -85,B 0,C 180,E1 -1183.313,E2 -1183.313} C_VEL
LIN {X 0,Y 594.442,Z 346.603,A -85,B 0,C 180,E1 -1183.352,E2 -1183.352} C_VEL
LIN {X 0,Y 594.498,Z 326.055,A -85,B 0,C 180,E1 -1186.131,E2 -1186.131} C_VEL
LIN {X 0,Y 594.609,Z 306.004,A -85,B 0,C 180,E1 -1188.878,E2 -1188.878} C_VEL
LIN {X 0,Y 594.774,Z 283.34,A -85,B 0,C 180,E1 -1192.035,E2 -1192.035} C_VEL
LIN {X 0,Y 594.668,Z 277.935,A -85,B 0,C 180,E1 -1192.804,E2 -1192.804} C_VEL
LIN {X 0,Y 594.392,Z 276.445,A -85,B 0,C 180,E1 -1193.059,E2 -1193.059} C_VEL
LIN {X 0,Y 594.366,Z 276.443,A -85,B 0,C 180,E1 -1195.194,E2 -1195.194} C_VEL
LIN {X 0,Y 594.372,Z 276.444,A -85,B 0,C 180,E1 -1197.524,E2 -1197.524} C_VEL
LIN {X 0,Y 594.389,Z 276.445,A -85,B 0,C 180,E1 -1200.328,E2 -1200.328} C_VEL
LIN {X 0,Y 594.378,Z 276.44,A -85,B 0,C 180,E1 -1202.95,E2 -1202.95} C_VEL
LIN {X 0,Y 594.349,Z 276.444,A -85,B 0,C 180,E1 -1205.409,E2 -1205.409} C_VEL
LIN {X 0,Y 594.386,Z 276.444,A -85,B 0,C 180,E1 -1207.94,E2 -1207.94} C_VEL
LIN {X 0,Y 594.376,Z 276.443,A -85,B 0,C 180,E1 -1210.822,E2 -1210.822} C_VEL
LIN {X 0,Y 594.365,Z 276.441,A -85,B 0,C 180,E1 -1213.299,E2 -1213.299} C_VEL
LIN {X 0,Y 594.356,Z 276.449,A -85,B 0,C 180,E1 -1216.161,E2 -1216.161} C_VEL
LIN {X 0,Y 594.378,Z 276.451,A -85,B 0,C 180,E1 -1218.536,E2 -1218.536} C_VEL
LIN {X 0,Y 594.381,Z 276.44,A -85,B 0,C 180,E1 -1221.295,E2 -1221.295} C_VEL
LIN {X 0,Y 594.388,Z 276.439,A -85,B 0,C 180,E1 -1223.758,E2 -1223.758} C_VEL
LIN {X 0,Y 594.376,Z 276.444,A -85,B 0,C 180,E1 -1226.238,E2 -1226.238} C_VEL
LIN {X 0,Y 594.383,Z 276.449,A -85,B 0,C 180,E1 -1228.65,E2 -1228.65} C_VEL
LIN {X 0,Y 594.372,Z 276.447,A -85,B 0,C 180,E1 -1231.042,E2 -1231.042} C_VEL
LIN {X 0,Y 594.382,Z 276.439,A -85,B 0,C 180,E1 -1233.975,E2 -1233.975} C_VEL
LIN {X 0,Y 594.38,Z 276.441,A -85,B 0,C 180,E1 -1236.295,E2 -1236.295} C_VEL
LIN {X 0,Y 594.387,Z 276.446,A -85,B 0,C 180,E1 -1239.224,E2 -1239.224} C_VEL
LIN {X 0,Y 594.341,Z 276.444,A -85,B 0,C 180,E1 -1242.095,E2 -1242.095} C_VEL
LIN {X 0,Y 594.355,Z 276.443,A -85,B 0,C 180,E1 -1244.219,E2 -1244.219} C_VEL
LIN {X 0,Y 594.358,Z 276.451,A -85,B 0,C 180,E1 -1247.017,E2 -1247.017} C_VEL
LIN {X 0,Y 594.373,Z 276.443,A -85,B 0,C 180,E1 -1249.784,E2 -1249.784} C_VEL
LIN {X 0,Y 594.388,Z 276.439,A -85,B 0,C 180,E1 -1252.527,E2 -1252.527} C_VEL
LIN {X 0,Y 594.396,Z 276.447,A -85,B 0,C 180,E1 -1255.252,E2 -1255.252} C_VEL
LIN {X 0,Y 594.365,Z 276.444,A -85,B 0,C 180,E1 -1257.967,E2 -1257.967} C_VEL
LIN {X 0,Y 594.382,Z 276.442,A -85,B 0,C 180,E1 -1260,E2 -1260} C_VEL
LIN {X 0,Y 594.382,Z 276.44,A -85,B 0,C 180,E1 -1262.711,E2 -1262.711} C_VEL
LIN {X 0,Y 594.389,Z 276.446,A -85,B 0,C 180,E1 -1265.428,E2 -1265.428} C_VEL
LIN {X 0,Y 594.364,Z 276.445,A -85,B 0,C 180,E1 -1268.157,E2 -1268.157} C_VEL
LIN {X 0,Y 594.36,Z 276.443,A -85,B 0,C 180,E1 -1271.067,E2 -1271.067} C_VEL
LIN {X 0,Y 594.368,Z 276.45,A -85,B 0,C 180,E1 -1273.679,E2 -1273.679} C_VEL
LIN {X 0,Y 594.328,Z 276.448,A -85,B 0,C 180,E1 -1275.304,E2 -1275.304} C_VEL
LIN {X 0,Y 593.666,Z 276.54,A -85,B 0,C 180,E1 -1275.87,E2 -1275.87} C_VEL
LIN {X 0,Y 590.82,Z 276.897,A -85,B 0,C 180,E1 -1276.788,E2 -1276.788} C_VEL
LIN {X 0,Y 588.413,Z 277.195,A -85,B 0,C 180,E1 -1277.526,E2 -1277.526} C_VEL
LIN {X 0,Y 587.38,Z 277.32,A -85,B 0,C 180,E1 -1278.096,E2 -1278.096} C_VEL
LIN {X 0,Y 587.296,Z 277.327,A -85,B 0,C 180,E1 -1278.289,E2 -1278.289} C_VEL
LIN {X 0,Y 587.318,Z 277.319,A -85,B 0,C 180,E1 -1281.038,E2 -1281.038} C_VEL
LIN {X 0,Y 587.304,Z 277.332,A -85,B 0,C 180,E1 -1284.008,E2 -1284.008} C_VEL
LIN {X 0,Y 587.288,Z 277.331,A -85,B 0,C 180,E1 -1286.281,E2 -1286.281} C_VEL
LIN {X 0,Y 587.29,Z 277.323,A -85,B 0,C 180,E1 -1289.125,E2 -1289.125} C_VEL
LIN {X 0,Y 587.33,Z 277.322,A -85,B 0,C 180,E1 -1291.835,E2 -1291.835} C_VEL
LIN {X 0,Y 587.322,Z 277.33,A -85,B 0,C 180,E1 -1294.346,E2 -1294.346} C_VEL
LIN {X 0,Y 587.298,Z 277.322,A -85,B 0,C 180,E1 -1297.611,E2 -1297.611} C_VEL
LIN {X 0,Y 587.278,Z 277.332,A -85,B 0,C 180,E1 -1300.258,E2 -1300.258} C_VEL
LIN {X 0,Y 587.272,Z 277.327,A -85,B 0,C 180,E1 -1303.115,E2 -1303.115} C_VEL
LIN {X 0,Y 587.281,Z 277.326,A -85,B 0,C 180,E1 -1306.046,E2 -1306.046} C_VEL
LIN {X 0,Y 587.28,Z 277.33,A -85,B 0,C 180,E1 -1308.932,E2 -1308.932} C_VEL
LIN {X 0,Y 587.261,Z 277.327,A -85,B 0,C 180,E1 -1311.516,E2 -1311.516} C_VEL
LIN {X 0,Y 587.247,Z 277.329,A -85,B 0,C 180,E1 -1314.097,E2 -1314.097} C_VEL
LIN {X 0,Y 587.273,Z 277.335,A -85,B 0,C 180,E1 -1316.899,E2 -1316.899} C_VEL
LIN {X 0,Y 587.271,Z 277.327,A -85,B 0,C 180,E1 -1319.502,E2 -1319.502} C_VEL
LIN {X 0,Y 587.298,Z 277.323,A -85,B 0,C 180,E1 -1322.318,E2 -1322.318} C_VEL
LIN {X 0,Y 587.286,Z 277.331,A -85,B 0,C 180,E1 -1325.238,E2 -1325.238} C_VEL
LIN {X 0,Y 587.304,Z 277.325,A -85,B 0,C 180,E1 -1327.484,E2 -1327.484} C_VEL
LIN {X 0,Y 587.311,Z 277.323,A -85,B 0,C 180,E1 -1329.694,E2 -1329.694} C_VEL
LIN {X 0,Y 587.281,Z 277.325,A -85,B 0,C 180,E1 -1331.871,E2 -1331.871} C_VEL
LIN {X 0,Y 587.293,Z 277.323,A -85,B 0,C 180,E1 -1334.023,E2 -1334.023} C_VEL
LIN {X 0,Y 587.328,Z 277.318,A -85,B 0,C 180,E1 -1336.152,E2 -1336.152} C_VEL
LIN {X 0,Y 587.343,Z 277.32,A -85,B 0,C 180,E1 -1338.961,E2 -1338.961} C_VEL
LIN {X 0,Y 587.321,Z 277.324,A -85,B 0,C 180,E1 -1341.742,E2 -1341.742} C_VEL
LIN {X 0,Y 587.323,Z 277.319,A -85,B 0,C 180,E1 -1344.505,E2 -1344.505} C_VEL
LIN {X 0,Y 587.357,Z 277.32,A -85,B 0,C 180,E1 -1347.255,E2 -1347.255} C_VEL
LIN {X 0,Y 587.382,Z 277.316,A -85,B 0,C 180,E1 -1349.998,E2 -1349.998} C_VEL
LIN {X 0,Y 587.343,Z 277.316,A -85,B 0,C 180,E1 -1352.741,E2 -1352.741} C_VEL
LIN {X 0,Y 587.338,Z 277.323,A -85,B 0,C 180,E1 -1355.491,E2 -1355.491} C_VEL
LIN {X 0,Y 587.339,Z 277.321,A -85,B 0,C 180,E1 -1358.253,E2 -1358.253} C_VEL
LIN {X 0,Y 587.297,Z 277.324,A -85,B 0,C 180,E1 -1361.106,E2 -1361.106} C_VEL
LIN {X 0,Y 587.347,Z 277.361,A -85,B 0,C 180,E1 -1363.094,E2 -1363.094} C_VEL
LIN {X 0,Y 587.442,Z 287.509,A -85,B 0,C 180,E1 -1364.902,E2 -1364.902} C_VEL
LIN {X 0,Y 587.35,Z 303.801,A -85,B 0,C 180,E1 -1367.762,E2 -1367.762} C_VEL
LIN {X 0,Y 587.363,Z 308.326,A -85,B 0,C 180,E1 -1368.551,E2 -1368.551} C_VEL
LIN {X 0,Y 587.866,Z 312.066,A -85,B 0,C 180,E1 -1368.624,E2 -1368.624} C_VEL
LIN {X 0,Y 587.708,Z 414.948,A -85,B 0,C 180,E1 -1369.9,E2 -1369.9} C_VEL
LIN {X 0,Y 587.673,Z 427.931,A -85,B 0,C 180,E1 -1370.197,E2 -1370.197} C_VEL
LIN {X 0,Y 587.609,Z 440.138,A -85,B 0,C 180,E1 -1370.611,E2 -1370.611} C_VEL
LIN {X 0,Y 587.532,Z 451.915,A -85,B 0,C 180,E1 -1371.148,E2 -1371.148} C_VEL
LIN {X 0,Y 587.426,Z 463.875,A -85,B 0,C 180,E1 -1371.859,E2 -1371.859} C_VEL
LIN {X 0,Y 587.378,Z 474.065,A -85,B 0,C 180,E1 -1372.619,E2 -1372.619} C_VEL
LIN {X 0,Y 587.336,Z 483.024,A -85,B 0,C 180,E1 -1373.441,E2 -1373.441} C_VEL
LIN {X 0,Y 587.302,Z 491.174,A -85,B 0,C 180,E1 -1374.334,E2 -1374.334} C_VEL
LIN {X 0,Y 587.234,Z 498.511,A -85,B 0,C 180,E1 -1375.327,E2 -1375.327} C_VEL
LIN {X 0,Y 587.202,Z 505.268,A -85,B 0,C 180,E1 -1376.472,E2 -1376.472} C_VEL
LIN {X 0,Y 587.159,Z 510.675,A -85,B 0,C 180,E1 -1377.656,E2 -1377.656} C_VEL
LIN {X 0,Y 587.158,Z 513.918,A -85,B 0,C 180,E1 -1378.601,E2 -1378.601} C_VEL
LIN {X 0,Y 587.127,Z 516.002,A -85,B 0,C 180,E1 -1379.387,E2 -1379.387} C_VEL
LIN {X 0,Y 587.145,Z 517.959,A -85,B 0,C 180,E1 -1380.478,E2 -1380.478} C_VEL
LIN {X 0,Y 587.12,Z 518.951,A -85,B 0,C 180,E1 -1381.8,E2 -1381.8} C_VEL
LIN {X 0,Y 587.128,Z 518.545,A -85,B 0,C 180,E1 -1383.08,E2 -1383.08} C_VEL
LIN {X 0,Y 587.131,Z 516.811,A -85,B 0,C 180,E1 -1384.316,E2 -1384.316} C_VEL
LIN {X 0,Y 587.143,Z 513.833,A -85,B 0,C 180,E1 -1385.516,E2 -1385.516} C_VEL
LIN {X 0,Y 587.199,Z 509.359,A -85,B 0,C 180,E1 -1386.752,E2 -1386.752} C_VEL
LIN {X 0,Y 587.184,Z 504.213,A -85,B 0,C 180,E1 -1387.818,E2 -1387.818} C_VEL
LIN {X 0,Y 587.255,Z 497.373,A -85,B 0,C 180,E1 -1388.932,E2 -1388.932} C_VEL
LIN {X 0,Y 587.293,Z 488.962,A -85,B 0,C 180,E1 -1390.015,E2 -1390.015} C_VEL
LIN {X 0,Y 587.362,Z 478.603,A -85,B 0,C 180,E1 -1391.078,E2 -1391.078} C_VEL
LIN {X 0,Y 587.403,Z 467.96,A -85,B 0,C 180,E1 -1391.946,E2 -1391.946} C_VEL
LIN {X 0,Y 587.492,Z 457.003,A -85,B 0,C 180,E1 -1392.662,E2 -1392.662} C_VEL
LIN {X 0,Y 587.591,Z 444.723,A -85,B 0,C 180,E1 -1393.286,E2 -1393.286} C_VEL
LIN {X 0,Y 587.657,Z 432.532,A -85,B 0,C 180,E1 -1393.754,E2 -1393.754} C_VEL
LIN {X 0,Y 587.718,Z 420.062,A -85,B 0,C 180,E1 -1394.091,E2 -1394.091} C_VEL
LIN {X 0,Y 587.76,Z 405.715,A -85,B 0,C 180,E1 -1394.318,E2 -1394.318} C_VEL
LIN {X 0,Y 587.784,Z 311.225,A -85,B 0,C 180,E1 -1395.478,E2 -1395.478} C_VEL
LIN {X 0,Y 587.332,Z 308.312,A -85,B 0,C 180,E1 -1395.542,E2 -1395.542} C_VEL
LIN {X 0,Y 587.447,Z 290.699,A -85,B 0,C 180,E1 -1398.624,E2 -1398.624} C_VEL
LIN {X 0,Y 587.419,Z 277.983,A -85,B 0,C 180,E1 -1400.883,E2 -1400.883} C_VEL
LIN {X 0,Y 587.308,Z 277.325,A -85,B 0,C 180,E1 -1401.053,E2 -1401.053} C_VEL
LIN {X 0,Y 587.314,Z 277.321,A -85,B 0,C 180,E1 -1403.288,E2 -1403.288} C_VEL
LIN {X 0,Y 587.335,Z 277.321,A -85,B 0,C 180,E1 -1405.778,E2 -1405.778} C_VEL
LIN {X 0,Y 587.317,Z 277.33,A -85,B 0,C 180,E1 -1408.229,E2 -1408.229} C_VEL
LIN {X 0,Y 587.31,Z 277.323,A -85,B 0,C 180,E1 -1410.862,E2 -1410.862} C_VEL
LIN {X 0,Y 587.326,Z 277.322,A -85,B 0,C 180,E1 -1413.813,E2 -1413.813} C_VEL
LIN {X 0,Y 587.279,Z 277.331,A -85,B 0,C 180,E1 -1416.739,E2 -1416.739} C_VEL
LIN {X 0,Y 587.279,Z 277.325,A -85,B 0,C 180,E1 -1419.693,E2 -1419.693} C_VEL
LIN {X 0,Y 587.31,Z 277.331,A -85,B 0,C 180,E1 -1422.593,E2 -1422.593} C_VEL
LIN {X 0,Y 587.308,Z 277.321,A -85,B 0,C 180,E1 -1425.738,E2 -1425.738} C_VEL
LIN {X 0,Y 587.335,Z 277.323,A -85,B 0,C 180,E1 -1428.962,E2 -1428.962} C_VEL
LIN {X 0,Y 587.308,Z 277.321,A -85,B 0,C 180,E1 -1431.744,E2 -1431.744} C_VEL
LIN {X 0,Y 587.326,Z 277.325,A -85,B 0,C 180,E1 -1434.507,E2 -1434.507} C_VEL
LIN {X 0,Y 587.326,Z 277.322,A -85,B 0,C 180,E1 -1437.256,E2 -1437.256} C_VEL
LIN {X 0,Y 587.314,Z 277.319,A -85,B 0,C 180,E1 -1440,E2 -1440} C_VEL
LIN {X 0,Y 587.338,Z 277.325,A -85,B 0,C 180,E1 -1442.743,E2 -1442.743} C_VEL
LIN {X 0,Y 587.328,Z 277.321,A -85,B 0,C 180,E1 -1445.493,E2 -1445.493} C_VEL
LIN {X 0,Y 587.319,Z 277.319,A -85,B 0,C 180,E1 -1448.256,E2 -1448.256} C_VEL
LIN {X 0,Y 587.372,Z 277.321,A -85,B 0,C 180,E1 -1451.176,E2 -1451.176} C_VEL
LIN {X 0,Y 587.31,Z 277.321,A -85,B 0,C 180,E1 -1454.263,E2 -1454.263} C_VEL
LIN {X 0,Y 587.311,Z 277.324,A -85,B 0,C 180,E1 -1456.823,E2 -1456.823} C_VEL
LIN {X 0,Y 587.309,Z 277.325,A -85,B 0,C 180,E1 -1459.576,E2 -1459.576} C_VEL
LIN {X 0,Y 587.325,Z 277.319,A -85,B 0,C 180,E1 -1462.514,E2 -1462.514} C_VEL
LIN {X 0,Y 587.315,Z 277.328,A -85,B 0,C 180,E1 -1465.518,E2 -1465.518} C_VEL
LIN {X 0,Y 587.31,Z 277.324,A -85,B 0,C 180,E1 -1467.82,E2 -1467.82} C_VEL
LIN {X 0,Y 587.312,Z 277.32,A -85,B 0,C 180,E1 -1470.517,E2 -1470.517} C_VEL
LIN {X 0,Y 587.315,Z 277.329,A -85,B 0,C 180,E1 -1473.398,E2 -1473.398} C_VEL
LIN {X 0,Y 587.324,Z 277.324,A -85,B 0,C 180,E1 -1475.898,E2 -1475.898} C_VEL
LIN {X 0,Y 587.307,Z 277.321,A -85,B 0,C 180,E1 -1478.481,E2 -1478.481} C_VEL
LIN {X 0,Y 587.333,Z 277.321,A -85,B 0,C 180,E1 -1481.157,E2 -1481.157} C_VEL
LIN {X 0,Y 587.3,Z 277.326,A -85,B 0,C 180,E1 -1484.118,E2 -1484.118} C_VEL
LIN {X 0,Y 587.311,Z 277.322,A -85,B 0,C 180,E1 -1487,E2 -1487} C_VEL
LIN {X 0,Y 587.307,Z 277.332,A -85,B 0,C 180,E1 -1489.751,E2 -1489.751} C_VEL
LIN {X 0,Y 587.33,Z 277.321,A -85,B 0,C 180,E1 -1492.397,E2 -1492.397} C_VEL
LIN {X 0,Y 587.331,Z 277.318,A -85,B 0,C 180,E1 -1494.95,E2 -1494.95} C_VEL
LIN {X 0,Y 587.324,Z 277.322,A -85,B 0,C 180,E1 -1497.425,E2 -1497.425} C_VEL
LIN {X 0,Y 587.332,Z 277.327,A -85,B 0,C 180,E1 -1499.835,E2 -1499.835} C_VEL
LIN {X 0,Y 587.337,Z 277.324,A -85,B 0,C 180,E1 -1502.31,E2 -1502.31} C_VEL
LIN {X 0,Y 587.327,Z 277.324,A -85,B 0,C 180,E1 -1504.487,E2 -1504.487} C_VEL
LIN {X 0,Y 587.351,Z 277.443,A -85,B 0,C 180,E1 -1506.824,E2 -1506.824} C_VEL
LIN {X 0,Y 587.851,Z 280.931,A -85,B 0,C 180,E1 -1507.346,E2 -1507.346} C_VEL
LIN {X 0,Y 587.704,Z 298.906,A -85,B 0,C 180,E1 -1509.895,E2 -1509.895} C_VEL
LIN {X 0,Y 587.563,Z 319.476,A -85,B 0,C 180,E1 -1512.764,E2 -1512.764} C_VEL
LIN {X 0,Y 587.447,Z 341.898,A -85,B 0,C 180,E1 -1515.844,E2 -1515.844} C_VEL
LIN {X 0,Y 587.406,Z 346.637,A -85,B 0,C 180,E1 -1516.489,E2 -1516.489} C_VEL
LIN {X 0,Y 587.884,Z 350.983,A -85,B 0,C 180,E1 -1516.567,E2 -1516.567} C_VEL
LIN {X 0,Y 587.722,Z 455.11,A -85,B 0,C 180,E1 -1517.858,E2 -1517.858} C_VEL
LIN {X 0,Y 587.671,Z 468.327,A -85,B 0,C 180,E1 -1518.163,E2 -1518.163} C_VEL
LIN {X 0,Y 587.618,Z 480.663,A -85,B 0,C 180,E1 -1518.586,E2 -1518.586} C_VEL
LIN {X 0,Y 587.548,Z 492.685,A -85,B 0,C 180,E1 -1519.144,E2 -1519.144} C_VEL
LIN {X 0,Y 587.441,Z 504.246,A -85,B 0,C 180,E1 -1519.839,E2 -1519.839} C_VEL
LIN {X 0,Y 587.391,Z 514.634,A -85,B 0,C 180,E1 -1520.621,E2 -1520.621} C_VEL
LIN {X 0,Y 587.308,Z 523.07,A -85,B 0,C 180,E1 -1521.4,E2 -1521.4} C_VEL
LIN {X 0,Y 587.272,Z 530.984,A -85,B 0,C 180,E1 -1522.266,E2 -1522.266} C_VEL
LIN {X 0,Y 587.229,Z 537.489,A -85,B 0,C 180,E1 -1523.129,E2 -1523.129} C_VEL
LIN {X 0,Y 587.236,Z 543.881,A -85,B 0,C 180,E1 -1524.164,E2 -1524.164} C_VEL
LIN {X 0,Y 587.147,Z 548.961,A -85,B 0,C 180,E1 -1525.196,E2 -1525.196} C_VEL
LIN {X 0,Y 587.212,Z 552.904,A -85,B 0,C 180,E1 -1526.228,E2 -1526.228} C_VEL
LIN {X 0,Y 587.132,Z 555.814,A -85,B 0,C 180,E1 -1527.258,E2 -1527.258} C_VEL
LIN {X 0,Y 587.139,Z 557.204,A -85,B 0,C 180,E1 -1527.944,E2 -1527.944} C_VEL
LIN {X 0,Y 587.14,Z 558.786,A -85,B 0,C 180,E1 -1529.316,E2 -1529.316} C_VEL
LIN {X 0,Y 587.137,Z 559,A -85,B 0,C 180,E1 -1530.002,E2 -1530.002} C_VEL
LIN {X 0,Y 587.147,Z 558.183,A -85,B 0,C 180,E1 -1531.374,E2 -1531.374} C_VEL
LIN {X 0,Y 587.139,Z 557.197,A -85,B 0,C 180,E1 -1532.06,E2 -1532.06} C_VEL
LIN {X 0,Y 587.132,Z 555.805,A -85,B 0,C 180,E1 -1532.746,E2 -1532.746} C_VEL
LIN {X 0,Y 587.213,Z 552.89,A -85,B 0,C 180,E1 -1533.776,E2 -1533.776} C_VEL
LIN {X 0,Y 587.147,Z 548.941,A -85,B 0,C 180,E1 -1534.808,E2 -1534.808} C_VEL
LIN {X 0,Y 587.217,Z 542.867,A -85,B 0,C 180,E1 -1536.013,E2 -1536.013} C_VEL
LIN {X 0,Y 587.247,Z 536.224,A -85,B 0,C 180,E1 -1537.048,E2 -1537.048} C_VEL
LIN {X 0,Y 587.298,Z 527.976,A -85,B 0,C 180,E1 -1538.085,E2 -1538.085} C_VEL
LIN {X 0,Y 587.358,Z 517.583,A -85,B 0,C 180,E1 -1539.124,E2 -1539.124} C_VEL
LIN {X 0,Y 587.432,Z 507.907,A -85,B 0,C 180,E1 -1539.905,E2 -1539.905} C_VEL
LIN {X 0,Y 587.519,Z 497.301,A -85,B 0,C 180,E1 -1540.6,E2 -1540.6} C_VEL
LIN {X 0,Y 587.595,Z 485.305,A -85,B 0,C 180,E1 -1541.215,E2 -1541.215} C_VEL
LIN {X 0,Y 587.617,Z 473.198,A -85,B 0,C 180,E1 -1541.687,E2 -1541.687} C_VEL
LIN {X 0,Y 587.677,Z 460.46,A -85,B 0,C 180,E1 -1542.038,E2 -1542.038} C_VEL
LIN {X 0,Y 587.747,Z 447.193,A -85,B 0,C 180,E1 -1542.255,E2 -1542.255} C_VEL
LIN {X 0,Y 587.714,Z 348.824,A -85,B 0,C 180,E1 -1543.464,E2 -1543.464} C_VEL
LIN {X 0,Y 587.393,Z 346.603,A -85,B 0,C 180,E1 -1543.516,E2 -1543.516} C_VEL
LIN {X 0,Y 587.47,Z 328.643,A -85,B 0,C 180,E1 -1545.972,E2 -1545.972} C_VEL
LIN {X 0,Y 587.633,Z 309.228,A -85,B 0,C 180,E1 -1548.659,E2 -1548.659} C_VEL
LIN {X 0,Y 587.804,Z 288.493,A -85,B 0,C 180,E1 -1551.576,E2 -1551.576} C_VEL
LIN {X 0,Y 587.806,Z 279.776,A -85,B 0,C 180,E1 -1552.821,E2 -1552.821} C_VEL
LIN {X 0,Y 587.324,Z 277.325,A -85,B 0,C 180,E1 -1553.207,E2 -1553.207} C_VEL
LIN {X 0,Y 587.328,Z 277.323,A -85,B 0,C 180,E1 -1555.517,E2 -1555.517} C_VEL
LIN {X 0,Y 587.343,Z 277.325,A -85,B 0,C 180,E1 -1557.818,E2 -1557.818} C_VEL
LIN {X 0,Y 587.339,Z 277.321,A -85,B 0,C 180,E1 -1560.51,E2 -1560.51} C_VEL
LIN {X 0,Y 587.334,Z 277.318,A -85,B 0,C 180,E1 -1563.397,E2 -1563.397} C_VEL
LIN {X 0,Y 587.291,Z 277.328,A -85,B 0,C 180,E1 -1565.9,E2 -1565.9} C_VEL
LIN {X 0,Y 587.328,Z 277.325,A -85,B 0,C 180,E1 -1568.479,E2 -1568.479} C_VEL
LIN {X 0,Y 587.336,Z 277.317,A -85,B 0,C 180,E1 -1571.156,E2 -1571.156} C_VEL
LIN {X 0,Y 587.309,Z 277.326,A -85,B 0,C 180,E1 -1574.111,E2 -1574.111} C_VEL
LIN {X 0,Y 587.311,Z 277.323,A -85,B 0,C 180,E1 -1576.993,E2 -1576.993} C_VEL
LIN {X 0,Y 587.314,Z 277.32,A -85,B 0,C 180,E1 -1579.745,E2 -1579.745} C_VEL
LIN {X 0,Y 587.34,Z 277.324,A -85,B 0,C 180,E1 -1582.392,E2 -1582.392} C_VEL
LIN {X 0,Y 587.319,Z 277.325,A -85,B 0,C 180,E1 -1584.944,E2 -1584.944} C_VEL
LIN {X 0,Y 587.331,Z 277.319,A -85,B 0,C 180,E1 -1587.42,E2 -1587.42} C_VEL
LIN {X 0,Y 587.339,Z 277.317,A -85,B 0,C 180,E1 -1589.83,E2 -1589.83} C_VEL
LIN {X 0,Y 587.329,Z 277.327,A -85,B 0,C 180,E1 -1592.954,E2 -1592.954} C_VEL
LIN {X 0,Y 587.342,Z 277.319,A -85,B 0,C 180,E1 -1595.419,E2 -1595.419} C_VEL
LIN {X 0,Y 587.31,Z 277.321,A -85,B 0,C 180,E1 -1598.225,E2 -1598.225} C_VEL
LIN {X 0,Y 587.336,Z 277.326,A -85,B 0,C 180,E1 -1601.151,E2 -1601.151} C_VEL
LIN {X 0,Y 587.31,Z 277.32,A -85,B 0,C 180,E1 -1604.024,E2 -1604.024} C_VEL
LIN {X 0,Y 587.346,Z 277.316,A -85,B 0,C 180,E1 -1606.154,E2 -1606.154} C_VEL
LIN {X 0,Y 587.335,Z 277.323,A -85,B 0,C 180,E1 -1608.962,E2 -1608.962} C_VEL
LIN {X 0,Y 587.331,Z 277.321,A -85,B 0,C 180,E1 -1611.744,E2 -1611.744} C_VEL
LIN {X 0,Y 587.345,Z 277.316,A -85,B 0,C 180,E1 -1614.507,E2 -1614.507} C_VEL
LIN {X 0,Y 587.375,Z 277.32,A -85,B 0,C 180,E1 -1617.257,E2 -1617.257} C_VEL
LIN {X 0,Y 587.352,Z 277.318,A -85,B 0,C 180,E1 -1620,E2 -1620} C_VEL
LIN {X 0,Y 587.35,Z 277.316,A -85,B 0,C 180,E1 -1622.743,E2 -1622.743} C_VEL
LIN {X 0,Y 587.35,Z 277.324,A -85,B 0,C 180,E1 -1625.493,E2 -1625.493} C_VEL
LIN {X 0,Y 587.324,Z 277.321,A -85,B 0,C 180,E1 -1628.256,E2 -1628.256} C_VEL
LIN {X 0,Y 587.333,Z 277.319,A -85,B 0,C 180,E1 -1631.134,E2 -1631.134} C_VEL
LIN {X 0,Y 587.338,Z 277.328,A -85,B 0,C 180,E1 -1633.846,E2 -1633.846} C_VEL
LIN {X 0,Y 587.301,Z 277.321,A -85,B 0,C 180,E1 -1636.804,E2 -1636.804} C_VEL
LIN {X 0,Y 587.296,Z 277.327,A -85,B 0,C 180,E1 -1638.289,E2 -1638.289} C_VEL
LIN {X 0,Y 586.64,Z 277.406,A -85,B 0,C 180,E1 -1638.861,E2 -1638.861} C_VEL
LIN {X 0,Y 583.823,Z 277.763,A -85,B 0,C 180,E1 -1639.79,E2 -1639.79} C_VEL
LIN {X 0,Y 581.424,Z 278.057,A -85,B 0,C 180,E1 -1640.537,E2 -1640.537} C_VEL
LIN {X 0,Y 580.368,Z 278.186,A -85,B 0,C 180,E1 -1641.113,E2 -1641.113} C_VEL
LIN {X 0,Y 580.269,Z 278.198,A -85,B 0,C 180,E1 -1641.308,E2 -1641.308} C_VEL
LIN {X 0,Y 580.279,Z 278.203,A -85,B 0,C 180,E1 -1644.317,E2 -1644.317} C_VEL
LIN {X 0,Y 580.227,Z 278.205,A -85,B 0,C 180,E1 -1646.626,E2 -1646.626} C_VEL
LIN {X 0,Y 580.246,Z 278.2,A -85,B 0,C 180,E1 -1649.302,E2 -1649.302} C_VEL
LIN {X 0,Y 580.286,Z 278.206,A -85,B 0,C 180,E1 -1652.202,E2 -1652.202} C_VEL
LIN {X 0,Y 580.263,Z 278.202,A -85,B 0,C 180,E1 -1654.698,E2 -1654.698} C_VEL
LIN {X 0,Y 580.257,Z 278.199,A -85,B 0,C 180,E1 -1657.272,E2 -1657.272} C_VEL
LIN {X 0,Y 580.258,Z 278.202,A -85,B 0,C 180,E1 -1659.936,E2 -1659.936} C_VEL
LIN {X 0,Y 580.24,Z 278.208,A -85,B 0,C 180,E1 -1662.71,E2 -1662.71} C_VEL
LIN {X 0,Y 580.231,Z 278.202,A -85,B 0,C 180,E1 -1665.613,E2 -1665.613} C_VEL
LIN {X 0,Y 580.23,Z 278.206,A -85,B 0,C 180,E1 -1668.227,E2 -1668.227} C_VEL
LIN {X 0,Y 580.23,Z 278.209,A -85,B 0,C 180,E1 -1670.962,E2 -1670.962} C_VEL
LIN {X 0,Y 580.223,Z 278.203,A -85,B 0,C 180,E1 -1673.593,E2 -1673.593} C_VEL
LIN {X 0,Y 580.234,Z 278.21,A -85,B 0,C 180,E1 -1676.695,E2 -1676.695} C_VEL
LIN {X 0,Y 580.238,Z 278.204,A -85,B 0,C 180,E1 -1679.421,E2 -1679.421} C_VEL
LIN {X 0,Y 580.241,Z 278.201,A -85,B 0,C 180,E1 -1682.153,E2 -1682.153} C_VEL
LIN {X 0,Y 580.229,Z 278.211,A -85,B 0,C 180,E1 -1684.916,E2 -1684.916} C_VEL
LIN {X 0,Y 580.28,Z 278.205,A -85,B 0,C 180,E1 -1687.196,E2 -1687.196} C_VEL
LIN {X 0,Y 580.265,Z 278.204,A -85,B 0,C 180,E1 -1689.436,E2 -1689.436} C_VEL
LIN {X 0,Y 580.242,Z 278.204,A -85,B 0,C 180,E1 -1691.643,E2 -1691.643} C_VEL
LIN {X 0,Y 580.252,Z 278.202,A -85,B 0,C 180,E1 -1693.824,E2 -1693.824} C_VEL
LIN {X 0,Y 580.293,Z 278.195,A -85,B 0,C 180,E1 -1695.981,E2 -1695.981} C_VEL
LIN {X 0,Y 580.312,Z 278.194,A -85,B 0,C 180,E1 -1698.826,E2 -1698.826} C_VEL
LIN {X 0,Y 580.295,Z 278.201,A -85,B 0,C 180,E1 -1701.642,E2 -1701.642} C_VEL
LIN {X 0,Y 580.293,Z 278.194,A -85,B 0,C 180,E1 -1704.438,E2 -1704.438} C_VEL
LIN {X 0,Y 580.322,Z 278.196,A -85,B 0,C 180,E1 -1707.221,E2 -1707.221} C_VEL
LIN {X 0,Y 580.351,Z 278.192,A -85,B 0,C 180,E1 -1709.998,E2 -1709.998} C_VEL
LIN {X 0,Y 580.311,Z 278.192,A -85,B 0,C 180,E1 -1712.774,E2 -1712.774} C_VEL
LIN {X 0,Y 580.306,Z 278.2,A -85,B 0,C 180,E1 -1715.557,E2 -1715.557} C_VEL
LIN {X 0,Y 580.307,Z 278.196,A -85,B 0,C 180,E1 -1718.354,E2 -1718.354} C_VEL
LIN {X 0,Y 580.264,Z 278.2,A -85,B 0,C 180,E1 -1721.171,E2 -1721.171} C_VEL
LIN {X 0,Y 580.313,Z 278.342,A -85,B 0,C 180,E1 -1723.033,E2 -1723.033} C_VEL
LIN {X 0,Y 580.429,Z 287.726,A -85,B 0,C 180,E1 -1724.727,E2 -1724.727} C_VEL
LIN {X 0,Y 580.352,Z 302.857,A -85,B 0,C 180,E1 -1727.419,E2 -1727.419} C_VEL
LIN {X 0,Y 580.323,Z 308.39,A -85,B 0,C 180,E1 -1728.395,E2 -1728.395} C_VEL
LIN {X 0,Y 580.963,Z 314.177,A -85,B 0,C 180,E1 -1728.488,E2 -1728.488} C_VEL
LIN {X 0,Y 580.792,Z 415.436,A -85,B 0,C 180,E1 -1729.762,E2 -1729.762} C_VEL
LIN {X 0,Y 580.714,Z 428.869,A -85,B 0,C 180,E1 -1730.081,E2 -1730.081} C_VEL
LIN {X 0,Y 580.645,Z 440.825,A -85,B 0,C 180,E1 -1730.499,E2 -1730.499} C_VEL
LIN {X 0,Y 580.551,Z 453.136,A -85,B 0,C 180,E1 -1731.082,E2 -1731.082} C_VEL
LIN {X 0,Y 580.424,Z 464.28,A -85,B 0,C 180,E1 -1731.762,E2 -1731.762} C_VEL
LIN {X 0,Y 580.341,Z 475.328,A -85,B 0,C 180,E1 -1732.608,E2 -1732.608} C_VEL
LIN {X 0,Y 580.301,Z 485.141,A -85,B 0,C 180,E1 -1733.553,E2 -1733.553} C_VEL
LIN {X 0,Y 580.2,Z 493.274,A -85,B 0,C 180,E1 -1734.509,E2 -1734.509} C_VEL
LIN {X 0,Y 580.144,Z 499.932,A -85,B 0,C 180,E1 -1735.467,E2 -1735.467} C_VEL
LIN {X 0,Y 580.126,Z 506.41,A -85,B 0,C 180,E1 -1736.626,E2 -1736.626} C_VEL
LIN {X 0,Y 580.066,Z 511.458,A -85,B 0,C 180,E1 -1737.815,E2 -1737.815} C_VEL
LIN {X 0,Y 580.067,Z 515.091,A -85,B 0,C 180,E1 -1738.984,E2 -1738.984} C_VEL
LIN {X 0,Y 580.039,Z 516.887,A -85,B 0,C 180,E1 -1739.782,E2 -1739.782} C_VEL
LIN {X 0,Y 580.056,Z 518.185,A -85,B 0,C 180,E1 -1740.656,E2 -1740.656} C_VEL
LIN {X 0,Y 580.03,Z 518.993,A -85,B 0,C 180,E1 -1741.987,E2 -1741.987} C_VEL
LIN {X 0,Y 580.047,Z 518.361,A -85,B 0,C 180,E1 -1743.277,E2 -1743.277} C_VEL
LIN {X 0,Y 580.04,Z 516.447,A -85,B 0,C 180,E1 -1744.521,E2 -1744.521} C_VEL
LIN {X 0,Y 580.054,Z 513.313,A -85,B 0,C 180,E1 -1745.73,E2 -1745.73} C_VEL
LIN {X 0,Y 580.098,Z 508.96,A -85,B 0,C 180,E1 -1746.907,E2 -1746.907} C_VEL
LIN {X 0,Y 580.157,Z 502.756,A -85,B 0,C 180,E1 -1748.151,E2 -1748.151} C_VEL
LIN {X 0,Y 580.183,Z 495.209,A -85,B 0,C 180,E1 -1749.323,E2 -1749.323} C_VEL
LIN {X 0,Y 580.294,Z 486.864,A -85,B 0,C 180,E1 -1750.353,E2 -1750.353} C_VEL
LIN {X 0,Y 580.337,Z 476.952,A -85,B 0,C 180,E1 -1751.337,E2 -1751.337} C_VEL
LIN {X 0,Y 580.437,Z 465.927,A -85,B 0,C 180,E1 -1752.214,E2 -1752.214} C_VEL
LIN {X 0,Y 580.508,Z 454.822,A -85,B 0,C 180,E1 -1752.915,E2 -1752.915} C_VEL
LIN {X 0,Y 580.617,Z 443.545,A -85,B 0,C 180,E1 -1753.476,E2 -1753.476} C_VEL
LIN {X 0,Y 580.69,Z 432.054,A -85,B 0,C 180,E1 -1753.912,E2 -1753.912} C_VEL
LIN {X 0,Y 580.764,Z 419.357,A -85,B 0,C 180,E1 -1754.252,E2 -1754.252} C_VEL
LIN {X 0,Y 580.815,Z 404.459,A -85,B 0,C 180,E1 -1754.483,E2 -1754.483} C_VEL
LIN {X 0,Y 580.825,Z 311.729,A -85,B 0,C 180,E1 -1755.635,E2 -1755.635} C_VEL
LIN {X 0,Y 580.301,Z 308.354,A -85,B 0,C 180,E1 -1755.702,E2 -1755.702} C_VEL
LIN {X 0,Y 580.419,Z 291.738,A -85,B 0,C 180,E1 -1758.645,E2 -1758.645} C_VEL
LIN {X 0,Y 580.381,Z 278.794,A -85,B 0,C 180,E1 -1760.973,E2 -1760.973} C_VEL
LIN {X 0,Y 580.266,Z 278.203,A -85,B 0,C 180,E1 -1761.131,E2 -1761.131} C_VEL
LIN {X 0,Y 580.288,Z 278.206,A -85,B 0,C 180,E1 -1764.229,E2 -1764.229} C_VEL
LIN {X 0,Y 580.253,Z 278.201,A -85,B 0,C 180,E1 -1766.973,E2 -1766.973} C_VEL
LIN {X 0,Y 580.266,Z 278.199,A -85,B 0,C 180,E1 -1769.423,E2 -1769.423} C_VEL
LIN {X 0,Y 580.272,Z 278.205,A -85,B 0,C 180,E1 -1772.134,E2 -1772.134} C_VEL
LIN {X 0,Y 580.269,Z 278.202,A -85,B 0,C 180,E1 -1774.918,E2 -1774.918} C_VEL
LIN {X 0,Y 580.23,Z 278.206,A -85,B 0,C 180,E1 -1777.946,E2 -1777.946} C_VEL
LIN {X 0,Y 580.264,Z 278.203,A -85,B 0,C 180,E1 -1780.912,E2 -1780.912} C_VEL
LIN {X 0,Y 580.228,Z 278.204,A -85,B 0,C 180,E1 -1783.824,E2 -1783.824} C_VEL
LIN {X 0,Y 580.228,Z 278.213,A -85,B 0,C 180,E1 -1786.695,E2 -1786.695} C_VEL
LIN {X 0,Y 580.253,Z 278.2,A -85,B 0,C 180,E1 -1789.532,E2 -1789.532} C_VEL
LIN {X 0,Y 580.284,Z 278.2,A -85,B 0,C 180,E1 -1792.344,E2 -1792.344} C_VEL
LIN {X 0,Y 580.285,Z 278.2,A -85,B 0,C 180,E1 -1795.137,E2 -1795.137} C_VEL
LIN {X 0,Y 580.271,Z 278.197,A -85,B 0,C 180,E1 -1797.918,E2 -1797.918} C_VEL
LIN {X 0,Y 580.326,Z 278.197,A -85,B 0,C 180,E1 -1800.694,E2 -1800.694} C_VEL
LIN {X 0,Y 580.255,Z 278.201,A -85,B 0,C 180,E1 -1803.472,E2 -1803.472} C_VEL
LIN {X 0,Y 580.29,Z 278.197,A -85,B 0,C 180,E1 -1805.56,E2 -1805.56} C_VEL
LIN {X 0,Y 580.284,Z 278.196,A -85,B 0,C 180,E1 -1808.357,E2 -1808.357} C_VEL
LIN {X 0,Y 580.325,Z 278.198,A -85,B 0,C 180,E1 -1811.234,E2 -1811.234} C_VEL
LIN {X 0,Y 580.26,Z 278.199,A -85,B 0,C 180,E1 -1814.341,E2 -1814.341} C_VEL
LIN {X 0,Y 580.265,Z 278.203,A -85,B 0,C 180,E1 -1816.919,E2 -1816.919} C_VEL
LIN {X 0,Y 580.267,Z 278.199,A -85,B 0,C 180,E1 -1819.824,E2 -1819.824} C_VEL
LIN {X 0,Y 580.303,Z 278.196,A -85,B 0,C 180,E1 -1822.802,E2 -1822.802} C_VEL
LIN {X 0,Y 580.267,Z 278.201,A -85,B 0,C 180,E1 -1825.85,E2 -1825.85} C_VEL
LIN {X 0,Y 580.269,Z 278.197,A -85,B 0,C 180,E1 -1828.187,E2 -1828.187} C_VEL
LIN {X 0,Y 580.261,Z 278.199,A -85,B 0,C 180,E1 -1830.702,E2 -1830.702} C_VEL
LIN {X 0,Y 580.279,Z 278.204,A -85,B 0,C 180,E1 -1833.323,E2 -1833.323} C_VEL
LIN {X 0,Y 580.292,Z 278.202,A -85,B 0,C 180,E1 -1835.772,E2 -1835.772} C_VEL
LIN {X 0,Y 580.274,Z 278.199,A -85,B 0,C 180,E1 -1838.148,E2 -1838.148} C_VEL
LIN {X 0,Y 580.297,Z 278.195,A -85,B 0,C 180,E1 -1840.844,E2 -1840.844} C_VEL
LIN {X 0,Y 580.259,Z 278.21,A -85,B 0,C 180,E1 -1843.66,E2 -1843.66} C_VEL
LIN {X 0,Y 580.263,Z 278.199,A -85,B 0,C 180,E1 -1846.611,E2 -1846.611} C_VEL
LIN {X 0,Y 580.296,Z 278.197,A -85,B 0,C 180,E1 -1849.163,E2 -1849.163} C_VEL
LIN {X 0,Y 580.272,Z 278.207,A -85,B 0,C 180,E1 -1851.93,E2 -1851.93} C_VEL
LIN {X 0,Y 580.286,Z 278.198,A -85,B 0,C 180,E1 -1854.461,E2 -1854.461} C_VEL
LIN {X 0,Y 580.275,Z 278.198,A -85,B 0,C 180,E1 -1856.979,E2 -1856.979} C_VEL
LIN {X 0,Y 580.295,Z 278.198,A -85,B 0,C 180,E1 -1859.43,E2 -1859.43} C_VEL
LIN {X 0,Y 580.305,Z 278.203,A -85,B 0,C 180,E1 -1862.14,E2 -1862.14} C_VEL
LIN {X 0,Y 580.297,Z 278.196,A -85,B 0,C 180,E1 -1864.924,E2 -1864.924} C_VEL
LIN {X 0,Y 580.321,Z 278.262,A -85,B 0,C 180,E1 -1866.662,E2 -1866.662} C_VEL
LIN {X 0,Y 580.961,Z 283.374,A -85,B 0,C 180,E1 -1867.417,E2 -1867.417} C_VEL
LIN {X 0,Y 580.763,Z 302.79,A -85,B 0,C 180,E1 -1870.198,E2 -1870.198} C_VEL
LIN {X 0,Y 580.559,Z 322.742,A -85,B 0,C 180,E1 -1873.008,E2 -1873.008} C_VEL
LIN {X 0,Y 580.428,Z 345.504,A -85,B 0,C 180,E1 -1876.168,E2 -1876.168} C_VEL
LIN {X 0,Y 580.408,Z 346.718,A -85,B 0,C 180,E1 -1876.334,E2 -1876.334} C_VEL
LIN {X 0,Y 580.959,Z 352.771,A -85,B 0,C 180,E1 -1876.426,E2 -1876.426} C_VEL
LIN {X 0,Y 580.783,Z 455.11,A -85,B 0,C 180,E1 -1877.711,E2 -1877.711} C_VEL
LIN {X 0,Y 580.715,Z 468.328,A -85,B 0,C 180,E1 -1878.02,E2 -1878.02} C_VEL
LIN {X 0,Y 580.626,Z 479.977,A -85,B 0,C 180,E1 -1878.42,E2 -1878.42} C_VEL
LIN {X 0,Y 580.573,Z 490.991,A -85,B 0,C 180,E1 -1878.924,E2 -1878.924} C_VEL
LIN {X 0,Y 580.484,Z 501.633,A -85,B 0,C 180,E1 -1879.54,E2 -1879.54} C_VEL
LIN {X 0,Y 580.372,Z 512.509,A -85,B 0,C 180,E1 -1880.33,E2 -1880.33} C_VEL
LIN {X 0,Y 580.303,Z 521.365,A -85,B 0,C 180,E1 -1881.12,E2 -1881.12} C_VEL
LIN {X 0,Y 580.22,Z 530.984,A -85,B 0,C 180,E1 -1882.171,E2 -1882.171} C_VEL
LIN {X 0,Y 580.154,Z 538.65,A -85,B 0,C 180,E1 -1883.221,E2 -1883.221} C_VEL
LIN {X 0,Y 580.139,Z 545.694,A -85,B 0,C 180,E1 -1884.441,E2 -1884.441} C_VEL
LIN {X 0,Y 580.107,Z 550.382,A -85,B 0,C 180,E1 -1885.486,E2 -1885.486} C_VEL
LIN {X 0,Y 580.122,Z 553.965,A -85,B 0,C 180,E1 -1886.53,E2 -1886.53} C_VEL
LIN {X 0,Y 580.043,Z 555.814,A -85,B 0,C 180,E1 -1887.225,E2 -1887.225} C_VEL
LIN {X 0,Y 580.038,Z 557.203,A -85,B 0,C 180,E1 -1887.919,E2 -1887.919} C_VEL
LIN {X 0,Y 580.04,Z 558.786,A -85,B 0,C 180,E1 -1889.308,E2 -1889.308} C_VEL
LIN {X 0,Y 580.037,Z 559,A -85,B 0,C 180,E1 -1890.002,E2 -1890.002} C_VEL
LIN {X 0,Y 580.046,Z 558.184,A -85,B 0,C 180,E1 -1891.391,E2 -1891.391} C_VEL
LIN {X 0,Y 580.038,Z 557.197,A -85,B 0,C 180,E1 -1892.085,E2 -1892.085} C_VEL
LIN {X 0,Y 580.043,Z 555.805,A -85,B 0,C 180,E1 -1892.78,E2 -1892.78} C_VEL
LIN {X 0,Y 580.11,Z 552.89,A -85,B 0,C 180,E1 -1893.823,E2 -1893.823} C_VEL
LIN {X 0,Y 580.053,Z 548.941,A -85,B 0,C 180,E1 -1894.867,E2 -1894.867} C_VEL
LIN {X 0,Y 580.141,Z 542.866,A -85,B 0,C 180,E1 -1896.087,E2 -1896.087} C_VEL
LIN {X 0,Y 580.186,Z 536.225,A -85,B 0,C 180,E1 -1897.134,E2 -1897.134} C_VEL
LIN {X 0,Y 580.247,Z 527.976,A -85,B 0,C 180,E1 -1898.184,E2 -1898.184} C_VEL
LIN {X 0,Y 580.333,Z 517.584,A -85,B 0,C 180,E1 -1899.235,E2 -1899.235} C_VEL
LIN {X 0,Y 580.437,Z 507.905,A -85,B 0,C 180,E1 -1900.025,E2 -1900.025} C_VEL
LIN {X 0,Y 580.532,Z 497.301,A -85,B 0,C 180,E1 -1900.729,E2 -1900.729} C_VEL
LIN {X 0,Y 580.614,Z 485.471,A -85,B 0,C 180,E1 -1901.345,E2 -1901.345} C_VEL
LIN {X 0,Y 580.672,Z 473.13,A -85,B 0,C 180,E1 -1901.831,E2 -1901.831} C_VEL
LIN {X 0,Y 580.757,Z 460.459,A -85,B 0,C 180,E1 -1902.184,E2 -1902.184} C_VEL
LIN {X 0,Y 580.836,Z 447.193,A -85,B 0,C 180,E1 -1902.404,E2 -1902.404} C_VEL
LIN {X 0,Y 580.799,Z 349.493,A -85,B 0,C 180,E1 -1903.619,E2 -1903.619} C_VEL
LIN {X 0,Y 580.398,Z 346.603,A -85,B 0,C 180,E1 -1903.682,E2 -1903.682} C_VEL
LIN {X 0,Y 580.537,Z 326.055,A -85,B 0,C 180,E1 -1906.53,E2 -1906.53} C_VEL
LIN {X 0,Y 580.74,Z 306.503,A -85,B 0,C 180,E1 -1909.275,E2 -1909.275} C_VEL
LIN {X 0,Y 580.952,Z 285.929,A -85,B 0,C 180,E1 -1912.213,E2 -1912.213} C_VEL
LIN {X 0,Y 580.788,Z 280.793,A -85,B 0,C 180,E1 -1912.963,E2 -1912.963} C_VEL
LIN {X 0,Y 580.277,Z 278.204,A -85,B 0,C 180,E1 -1913.379,E2 -1913.379} C_VEL
LIN {X 0,Y 580.281,Z 278.206,A -85,B 0,C 180,E1 -1915.85,E2 -1915.85} C_VEL
LIN {X 0,Y 580.298,Z 278.203,A -85,B 0,C 180,E1 -1918.186,E2 -1918.186} C_VEL
LIN {X 0,Y 580.287,Z 278.197,A -85,B 0,C 180,E1 -1920.694,E2 -1920.694} C_VEL
LIN {X 0,Y 580.304,Z 278.193,A -85,B 0,C 180,E1 -1923.316,E2 -1923.316} C_VEL
LIN {X 0,Y 580.246,Z 278.204,A -85,B 0,C 180,E1 -1925.756,E2 -1925.756} C_VEL
LIN {X 0,Y 580.288,Z 278.204,A -85,B 0,C 180,E1 -1928.146,E2 -1928.146} C_VEL
LIN {X 0,Y 580.298,Z 278.196,A -85,B 0,C 180,E1 -1930.843,E2 -1930.843} C_VEL
LIN {X 0,Y 580.271,Z 278.198,A -85,B 0,C 180,E1 -1933.658,E2 -1933.658} C_VEL
LIN {X 0,Y 580.271,Z 278.205,A -85,B 0,C 180,E1 -1936.609,E2 -1936.609} C_VEL
LIN {X 0,Y 580.295,Z 278.196,A -85,B 0,C 180,E1 -1939.156,E2 -1939.156} C_VEL
LIN {X 0,Y 580.286,Z 278.197,A -85,B 0,C 180,E1 -1941.926,E2 -1941.926} C_VEL
LIN {X 0,Y 580.279,Z 278.204,A -85,B 0,C 180,E1 -1944.454,E2 -1944.454} C_VEL
LIN {X 0,Y 580.284,Z 278.202,A -85,B 0,C 180,E1 -1946.975,E2 -1946.975} C_VEL
LIN {X 0,Y 580.301,Z 278.195,A -85,B 0,C 180,E1 -1949.425,E2 -1949.425} C_VEL
LIN {X 0,Y 580.289,Z 278.196,A -85,B 0,C 180,E1 -1952.141,E2 -1952.141} C_VEL
LIN {X 0,Y 580.299,Z 278.204,A -85,B 0,C 180,E1 -1954.92,E2 -1954.92} C_VEL
LIN {X 0,Y 580.26,Z 278.198,A -85,B 0,C 180,E1 -1957.947,E2 -1957.947} C_VEL
LIN {X 0,Y 580.307,Z 278.202,A -85,B 0,C 180,E1 -1960.914,E2 -1960.914} C_VEL
LIN {X 0,Y 580.263,Z 278.199,A -85,B 0,C 180,E1 -1963.825,E2 -1963.825} C_VEL
LIN {X 0,Y 580.312,Z 278.192,A -85,B 0,C 180,E1 -1965.983,E2 -1965.983} C_VEL
LIN {X 0,Y 580.318,Z 278.195,A -85,B 0,C 180,E1 -1968.827,E2 -1968.827} C_VEL
LIN {X 0,Y 580.302,Z 278.198,A -85,B 0,C 180,E1 -1971.644,E2 -1971.644} C_VEL
LIN {X 0,Y 580.309,Z 278.192,A -85,B 0,C 180,E1 -1974.44,E2 -1974.44} C_VEL
LIN {X 0,Y 580.339,Z 278.196,A -85,B 0,C 180,E1 -1977.223,E2 -1977.223} C_VEL
LIN {X 0,Y 580.323,Z 278.193,A -85,B 0,C 180,E1 -1980,E2 -1980} C_VEL
LIN {X 0,Y 580.319,Z 278.192,A -85,B 0,C 180,E1 -1982.777,E2 -1982.777} C_VEL
LIN {X 0,Y 580.313,Z 278.202,A -85,B 0,C 180,E1 -1985.56,E2 -1985.56} C_VEL
LIN {X 0,Y 580.293,Z 278.196,A -85,B 0,C 180,E1 -1988.357,E2 -1988.357} C_VEL
LIN {X 0,Y 580.286,Z 278.198,A -85,B 0,C 180,E1 -1991.191,E2 -1991.191} C_VEL
LIN {X 0,Y 580.292,Z 278.202,A -85,B 0,C 180,E1 -1994.018,E2 -1994.018} C_VEL
LIN {X 0,Y 580.276,Z 278.197,A -85,B 0,C 180,E1 -1996.907,E2 -1996.907} C_VEL
LIN {X 0,Y 580.267,Z 278.206,A -85,B 0,C 180,E1 -1999.824,E2 -1999.824} C_VEL
LIN {X 0,Y 580.269,Z 278.198,A -85,B 0,C 180,E1 -2001.308,E2 -2001.308} C_VEL
LIN {X 0,Y 579.563,Z 278.294,A -85,B 0,C 180,E1 -2001.887,E2 -2001.887} C_VEL
LIN {X 0,Y 576.686,Z 278.65,A -85,B 0,C 180,E1 -2002.827,E2 -2002.827} C_VEL
LIN {X 0,Y 574.29,Z 278.947,A -85,B 0,C 180,E1 -2003.584,E2 -2003.584} C_VEL
LIN {X 0,Y 573.282,Z 279.077,A -85,B 0,C 180,E1 -2004.167,E2 -2004.167} C_VEL
LIN {X 0,Y 573.21,Z 279.079,A -85,B 0,C 180,E1 -2004.365,E2 -2004.365} C_VEL
LIN {X 0,Y 573.174,Z 279.081,A -85,B 0,C 180,E1 -2006.98,E2 -2006.98} C_VEL
LIN {X 0,Y 573.225,Z 279.086,A -85,B 0,C 180,E1 -2010.178,E2 -2010.178} C_VEL
LIN {X 0,Y 573.241,Z 279.077,A -85,B 0,C 180,E1 -2012.646,E2 -2012.646} C_VEL
LIN {X 0,Y 573.175,Z 279.081,A -85,B 0,C 180,E1 -2015.19,E2 -2015.19} C_VEL
LIN {X 0,Y 573.208,Z 279.079,A -85,B 0,C 180,E1 -2017.81,E2 -2017.81} C_VEL
LIN {X 0,Y 573.194,Z 279.089,A -85,B 0,C 180,E1 -2020.53,E2 -2020.53} C_VEL
LIN {X 0,Y 573.182,Z 279.081,A -85,B 0,C 180,E1 -2023.365,E2 -2023.365} C_VEL
LIN {X 0,Y 573.189,Z 279.086,A -85,B 0,C 180,E1 -2026.337,E2 -2026.337} C_VEL
LIN {X 0,Y 573.185,Z 279.089,A -85,B 0,C 180,E1 -2028.539,E2 -2028.539} C_VEL
LIN {X 0,Y 573.169,Z 279.084,A -85,B 0,C 180,E1 -2031.293,E2 -2031.293} C_VEL
LIN {X 0,Y 573.174,Z 279.082,A -85,B 0,C 180,E1 -2033.946,E2 -2033.946} C_VEL
LIN {X 0,Y 573.182,Z 279.085,A -85,B 0,C 180,E1 -2036.512,E2 -2036.512} C_VEL
LIN {X 0,Y 573.196,Z 279.085,A -85,B 0,C 180,E1 -2039.124,E2 -2039.124} C_VEL
LIN {X 0,Y 573.196,Z 279.078,A -85,B 0,C 180,E1 -2041.982,E2 -2041.982} C_VEL
LIN {X 0,Y 573.192,Z 279.083,A -85,B 0,C 180,E1 -2044.586,E2 -2044.586} C_VEL
LIN {X 0,Y 573.216,Z 279.078,A -85,B 0,C 180,E1 -2047.661,E2 -2047.661} C_VEL
LIN {X 0,Y 573.232,Z 279.075,A -85,B 0,C 180,E1 -2049.922,E2 -2049.922} C_VEL
LIN {X 0,Y 573.219,Z 279.083,A -85,B 0,C 180,E1 -2053.005,E2 -2053.005} C_VEL
LIN {X 0,Y 573.243,Z 279.075,A -85,B 0,C 180,E1 -2055.805,E2 -2055.805} C_VEL
LIN {X 0,Y 573.269,Z 279.071,A -85,B 0,C 180,E1 -2058.744,E2 -2058.744} C_VEL
LIN {X 0,Y 573.24,Z 279.082,A -85,B 0,C 180,E1 -2061.538,E2 -2061.538} C_VEL
LIN {X 0,Y 573.263,Z 279.07,A -85,B 0,C 180,E1 -2064.37,E2 -2064.37} C_VEL
LIN {X 0,Y 573.307,Z 279.07,A -85,B 0,C 180,E1 -2067.89,E2 -2067.89} C_VEL
LIN {X 0,Y 573.319,Z 279.068,A -85,B 0,C 180,E1 -2069.998,E2 -2069.998} C_VEL
LIN {X 0,Y 573.279,Z 279.068,A -85,B 0,C 180,E1 -2072.808,E2 -2072.808} C_VEL
LIN {X 0,Y 573.274,Z 279.077,A -85,B 0,C 180,E1 -2075.626,E2 -2075.626} C_VEL
LIN {X 0,Y 573.25,Z 279.074,A -85,B 0,C 180,E1 -2078.457,E2 -2078.457} C_VEL
LIN {X 0,Y 573.233,Z 279.078,A -85,B 0,C 180,E1 -2081.31,E2 -2081.31} C_VEL
LIN {X 0,Y 573.25,Z 279.085,A -85,B 0,C 180,E1 -2082.926,E2 -2082.926} C_VEL
LIN {X 0,Y 573.433,Z 287.575,A -85,B 0,C 180,E1 -2084.482,E2 -2084.482} C_VEL
LIN {X 0,Y 573.342,Z 302.127,A -85,B 0,C 180,E1 -2087.105,E2 -2087.105} C_VEL
LIN {X 0,Y 573.276,Z 308.329,A -85,B 0,C 180,E1 -2088.213,E2 -2088.213} C_VEL
LIN {X 0,Y 574.061,Z 314.468,A -85,B 0,C 180,E1 -2088.326,E2 -2088.326} C_VEL
LIN {X 0,Y 573.85,Z 415.634,A -85,B 0,C 180,E1 -2089.615,E2 -2089.615} C_VEL
LIN {X 0,Y 573.783,Z 429.028,A -85,B 0,C 180,E1 -2089.939,E2 -2089.939} C_VEL
LIN {X 0,Y 573.669,Z 441.529,A -85,B 0,C 180,E1 -2090.385,E2 -2090.385} C_VEL
LIN {X 0,Y 573.569,Z 453.315,A -85,B 0,C 180,E1 -2090.957,E2 -2090.957} C_VEL
LIN {X 0,Y 573.411,Z 464.695,A -85,B 0,C 180,E1 -2091.664,E2 -2091.664} C_VEL
LIN {X 0,Y 573.324,Z 475.653,A -85,B 0,C 180,E1 -2092.52,E2 -2092.52} C_VEL
LIN {X 0,Y 573.249,Z 485.069,A -85,B 0,C 180,E1 -2093.439,E2 -2093.439} C_VEL
LIN {X 0,Y 573.129,Z 493.483,A -85,B 0,C 180,E1 -2094.443,E2 -2094.443} C_VEL
LIN {X 0,Y 573.059,Z 500.121,A -85,B 0,C 180,E1 -2095.415,E2 -2095.415} C_VEL
LIN {X 0,Y 573.035,Z 505.868,A -85,B 0,C 180,E1 -2096.451,E2 -2096.451} C_VEL
LIN {X 0,Y 573.007,Z 509.994,A -85,B 0,C 180,E1 -2097.379,E2 -2097.379} C_VEL
LIN {X 0,Y 572.974,Z 514.095,A -85,B 0,C 180,E1 -2098.574,E2 -2098.574} C_VEL
LIN {X 0,Y 572.962,Z 516.24,A -85,B 0,C 180,E1 -2099.437,E2 -2099.437} C_VEL
LIN {X 0,Y 572.961,Z 518.405,A -85,B 0,C 180,E1 -2100.837,E2 -2100.837} C_VEL
LIN {X 0,Y 572.94,Z 518.977,A -85,B 0,C 180,E1 -2102.178,E2 -2102.178} C_VEL
LIN {X 0,Y 572.965,Z 518.133,A -85,B 0,C 180,E1 -2103.497,E2 -2103.497} C_VEL
LIN {X 0,Y 572.952,Z 516.079,A -85,B 0,C 180,E1 -2104.73,E2 -2104.73} C_VEL
LIN {X 0,Y 572.992,Z 512.391,A -85,B 0,C 180,E1 -2106.062,E2 -2106.062} C_VEL
LIN {X 0,Y 573.015,Z 508.229,A -85,B 0,C 180,E1 -2107.134,E2 -2107.134} C_VEL
LIN {X 0,Y 573.075,Z 502.389,A -85,B 0,C 180,E1 -2108.291,E2 -2108.291} C_VEL
LIN {X 0,Y 573.132,Z 495.176,A -85,B 0,C 180,E1 -2109.418,E2 -2109.418} C_VEL
LIN {X 0,Y 573.215,Z 486.268,A -85,B 0,C 180,E1 -2110.521,E2 -2110.521} C_VEL
LIN {X 0,Y 573.295,Z 477.034,A -85,B 0,C 180,E1 -2111.445,E2 -2111.445} C_VEL
LIN {X 0,Y 573.411,Z 466.879,A -85,B 0,C 180,E1 -2112.272,E2 -2112.272} C_VEL
LIN {X 0,Y 573.515,Z 455.311,A -85,B 0,C 180,E1 -2113.021,E2 -2113.021} C_VEL
LIN {X 0,Y 573.675,Z 442.922,A -85,B 0,C 180,E1 -2113.644,E2 -2113.644} C_VEL
LIN {X 0,Y 573.756,Z 430.819,A -85,B 0,C 180,E1 -2114.099,E2 -2114.099} C_VEL
LIN {X 0,Y 573.846,Z 417.553,A -85,B 0,C 180,E1 -2114.437,E2 -2114.437} C_VEL
LIN {X 0,Y 573.884,Z 397.828,A -85,B 0,C 180,E1 -2114.719,E2 -2114.719} C_VEL
LIN {X 0,Y 573.997,Z 312.967,A -85,B 0,C 180,E1 -2115.785,E2 -2115.785} C_VEL
LIN {X 0,Y 573.28,Z 308.37,A -85,B 0,C 180,E1 -2115.869,E2 -2115.869} C_VEL
LIN {X 0,Y 573.399,Z 292.085,A -85,B 0,C 180,E1 -2118.792,E2 -2118.792} C_VEL
LIN {X 0,Y 573.44,Z 280.695,A -85,B 0,C 180,E1 -2120.863,E2 -2120.863} C_VEL
LIN {X 0,Y 573.243,Z 279.078,A -85,B 0,C 180,E1 -2121.186,E2 -2121.186} C_VEL
LIN {X 0,Y 573.225,Z 279.084,A -85,B 0,C 180,E1 -2124.007,E2 -2124.007} C_VEL
LIN {X 0,Y 573.241,Z 279.08,A -85,B 0,C 180,E1 -2126.516,E2 -2126.516} C_VEL
LIN {X 0,Y 573.201,Z 279.079,A -85,B 0,C 180,E1 -2129.111,E2 -2129.111} C_VEL
LIN {X 0,Y 573.217,Z 279.081,A -85,B 0,C 180,E1 -2131.965,E2 -2131.965} C_VEL
LIN {X 0,Y 573.218,Z 279.085,A -85,B 0,C 180,E1 -2134.588,E2 -2134.588} C_VEL
LIN {X 0,Y 573.191,Z 279.081,A -85,B 0,C 180,E1 -2137.66,E2 -2137.66} C_VEL
LIN {X 0,Y 573.223,Z 279.083,A -85,B 0,C 180,E1 -2140.726,E2 -2140.726} C_VEL
LIN {X 0,Y 573.198,Z 279.079,A -85,B 0,C 180,E1 -2143.62,E2 -2143.62} C_VEL
LIN {X 0,Y 573.186,Z 279.09,A -85,B 0,C 180,E1 -2146.528,E2 -2146.528} C_VEL
LIN {X 0,Y 573.225,Z 279.076,A -85,B 0,C 180,E1 -2149.403,E2 -2149.403} C_VEL
LIN {X 0,Y 573.233,Z 279.077,A -85,B 0,C 180,E1 -2152.249,E2 -2152.249} C_VEL
LIN {X 0,Y 573.258,Z 279.076,A -85,B 0,C 180,E1 -2155.077,E2 -2155.077} C_VEL
LIN {X 0,Y 573.243,Z 279.073,A -85,B 0,C 180,E1 -2157.892,E2 -2157.892} C_VEL
LIN {X 0,Y 573.294,Z 279.073,A -85,B 0,C 180,E1 -2160.702,E2 -2160.702} C_VEL
LIN {X 0,Y 573.204,Z 279.079,A -85,B 0,C 180,E1 -2163.515,E2 -2163.515} C_VEL
LIN {X 0,Y 573.253,Z 279.073,A -85,B 0,C 180,E1 -2165.629,E2 -2165.629} C_VEL
LIN {X 0,Y 573.257,Z 279.072,A -85,B 0,C 180,E1 -2168.46,E2 -2168.46} C_VEL
LIN {X 0,Y 573.269,Z 279.075,A -85,B 0,C 180,E1 -2171.312,E2 -2171.312} C_VEL
LIN {X 0,Y 573.226,Z 279.076,A -85,B 0,C 180,E1 -2174.427,E2 -2174.427} C_VEL
LIN {X 0,Y 573.225,Z 279.084,A -85,B 0,C 180,E1 -2177.113,E2 -2177.113} C_VEL
LIN {X 0,Y 573.216,Z 279.075,A -85,B 0,C 180,E1 -2180.078,E2 -2180.078} C_VEL
LIN {X 0,Y 573.259,Z 279.079,A -85,B 0,C 180,E1 -2183.165,E2 -2183.165} C_VEL
LIN {X 0,Y 573.252,Z 279.072,A -85,B 0,C 180,E1 -2186.19,E2 -2186.19} C_VEL
LIN {X 0,Y 573.213,Z 279.076,A -85,B 0,C 180,E1 -2188.566,E2 -2188.566} C_VEL
LIN {X 0,Y 573.204,Z 279.081,A -85,B 0,C 180,E1 -2190.995,E2 -2190.995} C_VEL
LIN {X 0,Y 573.244,Z 279.083,A -85,B 0,C 180,E1 -2193.531,E2 -2193.531} C_VEL
LIN {X 0,Y 573.237,Z 279.077,A -85,B 0,C 180,E1 -2196.05,E2 -2196.05} C_VEL
LIN {X 0,Y 573.225,Z 279.075,A -85,B 0,C 180,E1 -2198.703,E2 -2198.703} C_VEL
LIN {X 0,Y 573.23,Z 279.082,A -85,B 0,C 180,E1 -2201.457,E2 -2201.457} C_VEL
LIN {X 0,Y 573.206,Z 279.08,A -85,B 0,C 180,E1 -2204.337,E2 -2204.337} C_VEL
LIN {X 0,Y 573.232,Z 279.079,A -85,B 0,C 180,E1 -2207.36,E2 -2207.36} C_VEL
LIN {X 0,Y 573.228,Z 279.077,A -85,B 0,C 180,E1 -2210.398,E2 -2210.398} C_VEL
LIN {X 0,Y 573.235,Z 279.075,A -85,B 0,C 180,E1 -2213.082,E2 -2213.082} C_VEL
LIN {X 0,Y 573.256,Z 279.079,A -85,B 0,C 180,E1 -2215.676,E2 -2215.676} C_VEL
LIN {X 0,Y 573.234,Z 279.082,A -85,B 0,C 180,E1 -2218.189,E2 -2218.189} C_VEL
LIN {X 0,Y 573.255,Z 279.074,A -85,B 0,C 180,E1 -2220.639,E2 -2220.639} C_VEL
LIN {X 0,Y 573.259,Z 279.075,A -85,B 0,C 180,E1 -2223.504,E2 -2223.504} C_VEL
LIN {X 0,Y 573.271,Z 279.078,A -85,B 0,C 180,E1 -2226.529,E2 -2226.529} C_VEL
LIN {X 0,Y 574.008,Z 284.397,A -85,B 0,C 180,E1 -2227.318,E2 -2227.318} C_VEL
LIN {X 0,Y 573.827,Z 302.79,A -85,B 0,C 180,E1 -2229.948,E2 -2229.948} C_VEL
LIN {X 0,Y 573.585,Z 323.382,A -85,B 0,C 180,E1 -2232.885,E2 -2232.885} C_VEL
LIN {X 0,Y 573.427,Z 344.21,A -85,B 0,C 180,E1 -2235.814,E2 -2235.814} C_VEL
LIN {X 0,Y 573.409,Z 346.718,A -85,B 0,C 180,E1 -2236.164,E2 -2236.164} C_VEL
LIN {X 0,Y 574.059,Z 352.771,A -85,B 0,C 180,E1 -2236.259,E2 -2236.259} C_VEL
LIN {X 0,Y 573.859,Z 455.11,A -85,B 0,C 180,E1 -2237.56,E2 -2237.56} C_VEL
LIN {X 0,Y 573.791,Z 468.327,A -85,B 0,C 180,E1 -2237.873,E2 -2237.873} C_VEL
LIN {X 0,Y 573.678,Z 480.454,A -85,B 0,C 180,E1 -2238.297,E2 -2238.297} C_VEL
LIN {X 0,Y 573.576,Z 492.682,A -85,B 0,C 180,E1 -2238.876,E2 -2238.876} C_VEL
LIN {X 0,Y 573.436,Z 504.245,A -85,B 0,C 180,E1 -2239.588,E2 -2239.588} C_VEL
LIN {X 0,Y 573.327,Z 514.637,A -85,B 0,C 180,E1 -2240.388,E2 -2240.388} C_VEL
LIN {X 0,Y 573.237,Z 523.097,A -85,B 0,C 180,E1 -2241.187,E2 -2241.187} C_VEL
LIN {X 0,Y 573.159,Z 530.984,A -85,B 0,C 180,E1 -2242.074,E2 -2242.074} C_VEL
LIN {X 0,Y 573.077,Z 538.907,A -85,B 0,C 180,E1 -2243.178,E2 -2243.178} C_VEL
LIN {X 0,Y 573.07,Z 545.694,A -85,B 0,C 180,E1 -2244.372,E2 -2244.372} C_VEL
LIN {X 0,Y 573.028,Z 550.383,A -85,B 0,C 180,E1 -2245.43,E2 -2245.43} C_VEL
LIN {X 0,Y 573.022,Z 553.965,A -85,B 0,C 180,E1 -2246.487,E2 -2246.487} C_VEL
LIN {X 0,Y 572.959,Z 555.814,A -85,B 0,C 180,E1 -2247.19,E2 -2247.19} C_VEL
LIN {X 0,Y 572.946,Z 558.188,A -85,B 0,C 180,E1 -2248.597,E2 -2248.597} C_VEL
LIN {X 0,Y 572.938,Z 559,A -85,B 0,C 180,E1 -2250.002,E2 -2250.002} C_VEL
LIN {X 0,Y 572.946,Z 558.184,A -85,B 0,C 180,E1 -2251.408,E2 -2251.408} C_VEL
LIN {X 0,Y 572.938,Z 557.196,A -85,B 0,C 180,E1 -2252.111,E2 -2252.111} C_VEL
LIN {X 0,Y 572.959,Z 555.805,A -85,B 0,C 180,E1 -2252.814,E2 -2252.814} C_VEL
LIN {X 0,Y 573.015,Z 552.889,A -85,B 0,C 180,E1 -2253.87,E2 -2253.87} C_VEL
